   // UNICODE_TO_GBK[2130] := 16#4F5C;
   // UNICODE_TO_GBK[2131] := 16#D7F7;
   // UNICODE_TO_GBK[2132] := 16#4F5D;
   // UNICODE_TO_GBK[2133] := 16#D8FE;
   // UNICODE_TO_GBK[2134] := 16#4F5E;
   // UNICODE_TO_GBK[2135] := 16#D8FA;
   // UNICODE_TO_GBK[2136] := 16#4F5F;
   // UNICODE_TO_GBK[2137] := 16#D9A1;
   // UNICODE_TO_GBK[2138] := 16#4F60;
   // UNICODE_TO_GBK[2139] := 16#C4E3;
   // UNICODE_TO_GBK[2140] := 16#4F61;
   // UNICODE_TO_GBK[2141] := 16#81D9;
   // UNICODE_TO_GBK[2142] := 16#4F62;
   // UNICODE_TO_GBK[2143] := 16#81DA;
   // UNICODE_TO_GBK[2144] := 16#4F63;
   // UNICODE_TO_GBK[2145] := 16#D3B6;
   // UNICODE_TO_GBK[2146] := 16#4F64;
   // UNICODE_TO_GBK[2147] := 16#D8F4;
   // UNICODE_TO_GBK[2148] := 16#4F65;
   // UNICODE_TO_GBK[2149] := 16#D9DD;
   // UNICODE_TO_GBK[2150] := 16#4F66;
   // UNICODE_TO_GBK[2151] := 16#81DB;
   // UNICODE_TO_GBK[2152] := 16#4F67;
   // UNICODE_TO_GBK[2153] := 16#D8FB;
   // UNICODE_TO_GBK[2154] := 16#4F68;
   // UNICODE_TO_GBK[2155] := 16#81DC;
   // UNICODE_TO_GBK[2156] := 16#4F69;
   // UNICODE_TO_GBK[2157] := 16#C5E5;
   // UNICODE_TO_GBK[2158] := 16#4F6A;
   // UNICODE_TO_GBK[2159] := 16#81DD;
   // UNICODE_TO_GBK[2160] := 16#4F6B;
   // UNICODE_TO_GBK[2161] := 16#81DE;
   // UNICODE_TO_GBK[2162] := 16#4F6C;
   // UNICODE_TO_GBK[2163] := 16#C0D0;
   // UNICODE_TO_GBK[2164] := 16#4F6D;
   // UNICODE_TO_GBK[2165] := 16#81DF;
   // UNICODE_TO_GBK[2166] := 16#4F6E;
   // UNICODE_TO_GBK[2167] := 16#81E0;
   // UNICODE_TO_GBK[2168] := 16#4F6F;
   // UNICODE_TO_GBK[2169] := 16#D1F0;
   // UNICODE_TO_GBK[2170] := 16#4F70;
   // UNICODE_TO_GBK[2171] := 16#B0DB;
   // UNICODE_TO_GBK[2172] := 16#4F71;
   // UNICODE_TO_GBK[2173] := 16#81E1;
   // UNICODE_TO_GBK[2174] := 16#4F72;
   // UNICODE_TO_GBK[2175] := 16#81E2;
   // UNICODE_TO_GBK[2176] := 16#4F73;
   // UNICODE_TO_GBK[2177] := 16#BCD1;
   // UNICODE_TO_GBK[2178] := 16#4F74;
   // UNICODE_TO_GBK[2179] := 16#D9A6;
   // UNICODE_TO_GBK[2180] := 16#4F75;
   // UNICODE_TO_GBK[2181] := 16#81E3;
   // UNICODE_TO_GBK[2182] := 16#4F76;
   // UNICODE_TO_GBK[2183] := 16#D9A5;
   // UNICODE_TO_GBK[2184] := 16#4F77;
   // UNICODE_TO_GBK[2185] := 16#81E4;
   // UNICODE_TO_GBK[2186] := 16#4F78;
   // UNICODE_TO_GBK[2187] := 16#81E5;
   // UNICODE_TO_GBK[2188] := 16#4F79;
   // UNICODE_TO_GBK[2189] := 16#81E6;
   // UNICODE_TO_GBK[2190] := 16#4F7A;
   // UNICODE_TO_GBK[2191] := 16#81E7;
   // UNICODE_TO_GBK[2192] := 16#4F7B;
   // UNICODE_TO_GBK[2193] := 16#D9AC;
   // UNICODE_TO_GBK[2194] := 16#4F7C;
   // UNICODE_TO_GBK[2195] := 16#D9AE;
   // UNICODE_TO_GBK[2196] := 16#4F7D;
   // UNICODE_TO_GBK[2197] := 16#81E8;
   // UNICODE_TO_GBK[2198] := 16#4F7E;
   // UNICODE_TO_GBK[2199] := 16#D9AB;
   // UNICODE_TO_GBK[2200] := 16#4F7F;
   // UNICODE_TO_GBK[2201] := 16#CAB9;
   // UNICODE_TO_GBK[2202] := 16#4F80;
   // UNICODE_TO_GBK[2203] := 16#81E9;
   // UNICODE_TO_GBK[2204] := 16#4F81;
   // UNICODE_TO_GBK[2205] := 16#81EA;
   // UNICODE_TO_GBK[2206] := 16#4F82;
   // UNICODE_TO_GBK[2207] := 16#81EB;
   // UNICODE_TO_GBK[2208] := 16#4F83;
   // UNICODE_TO_GBK[2209] := 16#D9A9;
   // UNICODE_TO_GBK[2210] := 16#4F84;
   // UNICODE_TO_GBK[2211] := 16#D6B6;
   // UNICODE_TO_GBK[2212] := 16#4F85;
   // UNICODE_TO_GBK[2213] := 16#81EC;
   // UNICODE_TO_GBK[2214] := 16#4F86;
   // UNICODE_TO_GBK[2215] := 16#81ED;
   // UNICODE_TO_GBK[2216] := 16#4F87;
   // UNICODE_TO_GBK[2217] := 16#81EE;
   // UNICODE_TO_GBK[2218] := 16#4F88;
   // UNICODE_TO_GBK[2219] := 16#B3DE;
   // UNICODE_TO_GBK[2220] := 16#4F89;
   // UNICODE_TO_GBK[2221] := 16#D9A8;
   // UNICODE_TO_GBK[2222] := 16#4F8A;
   // UNICODE_TO_GBK[2223] := 16#81EF;
   // UNICODE_TO_GBK[2224] := 16#4F8B;
   // UNICODE_TO_GBK[2225] := 16#C0FD;
   // UNICODE_TO_GBK[2226] := 16#4F8C;
   // UNICODE_TO_GBK[2227] := 16#81F0;
   // UNICODE_TO_GBK[2228] := 16#4F8D;
   // UNICODE_TO_GBK[2229] := 16#CACC;
   // UNICODE_TO_GBK[2230] := 16#4F8E;
   // UNICODE_TO_GBK[2231] := 16#81F1;
   // UNICODE_TO_GBK[2232] := 16#4F8F;
   // UNICODE_TO_GBK[2233] := 16#D9AA;
   // UNICODE_TO_GBK[2234] := 16#4F90;
   // UNICODE_TO_GBK[2235] := 16#81F2;
   // UNICODE_TO_GBK[2236] := 16#4F91;
   // UNICODE_TO_GBK[2237] := 16#D9A7;
   // UNICODE_TO_GBK[2238] := 16#4F92;
   // UNICODE_TO_GBK[2239] := 16#81F3;
   // UNICODE_TO_GBK[2240] := 16#4F93;
   // UNICODE_TO_GBK[2241] := 16#81F4;
   // UNICODE_TO_GBK[2242] := 16#4F94;
   // UNICODE_TO_GBK[2243] := 16#D9B0;
   // UNICODE_TO_GBK[2244] := 16#4F95;
   // UNICODE_TO_GBK[2245] := 16#81F5;
   // UNICODE_TO_GBK[2246] := 16#4F96;
   // UNICODE_TO_GBK[2247] := 16#81F6;
   // UNICODE_TO_GBK[2248] := 16#4F97;
   // UNICODE_TO_GBK[2249] := 16#B6B1;
   // UNICODE_TO_GBK[2250] := 16#4F98;
   // UNICODE_TO_GBK[2251] := 16#81F7;
   // UNICODE_TO_GBK[2252] := 16#4F99;
   // UNICODE_TO_GBK[2253] := 16#81F8;
   // UNICODE_TO_GBK[2254] := 16#4F9A;
   // UNICODE_TO_GBK[2255] := 16#81F9;
   // UNICODE_TO_GBK[2256] := 16#4F9B;
   // UNICODE_TO_GBK[2257] := 16#B9A9;
   // UNICODE_TO_GBK[2258] := 16#4F9C;
   // UNICODE_TO_GBK[2259] := 16#81FA;
   // UNICODE_TO_GBK[2260] := 16#4F9D;
   // UNICODE_TO_GBK[2261] := 16#D2C0;
   // UNICODE_TO_GBK[2262] := 16#4F9E;
   // UNICODE_TO_GBK[2263] := 16#81FB;
   // UNICODE_TO_GBK[2264] := 16#4F9F;
   // UNICODE_TO_GBK[2265] := 16#81FC;
   // UNICODE_TO_GBK[2266] := 16#4FA0;
   // UNICODE_TO_GBK[2267] := 16#CFC0;
   // UNICODE_TO_GBK[2268] := 16#4FA1;
   // UNICODE_TO_GBK[2269] := 16#81FD;
   // UNICODE_TO_GBK[2270] := 16#4FA2;
   // UNICODE_TO_GBK[2271] := 16#81FE;
   // UNICODE_TO_GBK[2272] := 16#4FA3;
   // UNICODE_TO_GBK[2273] := 16#C2C2;
   // UNICODE_TO_GBK[2274] := 16#4FA4;
   // UNICODE_TO_GBK[2275] := 16#8240;
   // UNICODE_TO_GBK[2276] := 16#4FA5;
   // UNICODE_TO_GBK[2277] := 16#BDC4;
   // UNICODE_TO_GBK[2278] := 16#4FA6;
   // UNICODE_TO_GBK[2279] := 16#D5EC;
   // UNICODE_TO_GBK[2280] := 16#4FA7;
   // UNICODE_TO_GBK[2281] := 16#B2E0;
   // UNICODE_TO_GBK[2282] := 16#4FA8;
   // UNICODE_TO_GBK[2283] := 16#C7C8;
   // UNICODE_TO_GBK[2284] := 16#4FA9;
   // UNICODE_TO_GBK[2285] := 16#BFEB;
   // UNICODE_TO_GBK[2286] := 16#4FAA;
   // UNICODE_TO_GBK[2287] := 16#D9AD;
   // UNICODE_TO_GBK[2288] := 16#4FAB;
   // UNICODE_TO_GBK[2289] := 16#8241;
   // UNICODE_TO_GBK[2290] := 16#4FAC;
   // UNICODE_TO_GBK[2291] := 16#D9AF;
   // UNICODE_TO_GBK[2292] := 16#4FAD;
   // UNICODE_TO_GBK[2293] := 16#8242;
   // UNICODE_TO_GBK[2294] := 16#4FAE;
   // UNICODE_TO_GBK[2295] := 16#CEEA;
   // UNICODE_TO_GBK[2296] := 16#4FAF;
   // UNICODE_TO_GBK[2297] := 16#BAEE;
   // UNICODE_TO_GBK[2298] := 16#4FB0;
   // UNICODE_TO_GBK[2299] := 16#8243;
   // UNICODE_TO_GBK[2300] := 16#4FB1;
   // UNICODE_TO_GBK[2301] := 16#8244;
   // UNICODE_TO_GBK[2302] := 16#4FB2;
   // UNICODE_TO_GBK[2303] := 16#8245;
   // UNICODE_TO_GBK[2304] := 16#4FB3;
   // UNICODE_TO_GBK[2305] := 16#8246;
   // UNICODE_TO_GBK[2306] := 16#4FB4;
   // UNICODE_TO_GBK[2307] := 16#8247;
   // UNICODE_TO_GBK[2308] := 16#4FB5;
   // UNICODE_TO_GBK[2309] := 16#C7D6;
   // UNICODE_TO_GBK[2310] := 16#4FB6;
   // UNICODE_TO_GBK[2311] := 16#8248;
   // UNICODE_TO_GBK[2312] := 16#4FB7;
   // UNICODE_TO_GBK[2313] := 16#8249;
   // UNICODE_TO_GBK[2314] := 16#4FB8;
   // UNICODE_TO_GBK[2315] := 16#824A;
   // UNICODE_TO_GBK[2316] := 16#4FB9;
   // UNICODE_TO_GBK[2317] := 16#824B;
   // UNICODE_TO_GBK[2318] := 16#4FBA;
   // UNICODE_TO_GBK[2319] := 16#824C;
   // UNICODE_TO_GBK[2320] := 16#4FBB;
   // UNICODE_TO_GBK[2321] := 16#824D;
   // UNICODE_TO_GBK[2322] := 16#4FBC;
   // UNICODE_TO_GBK[2323] := 16#824E;
   // UNICODE_TO_GBK[2324] := 16#4FBD;
   // UNICODE_TO_GBK[2325] := 16#824F;
   // UNICODE_TO_GBK[2326] := 16#4FBE;
   // UNICODE_TO_GBK[2327] := 16#8250;
   // UNICODE_TO_GBK[2328] := 16#4FBF;
   // UNICODE_TO_GBK[2329] := 16#B1E3;
   // UNICODE_TO_GBK[2330] := 16#4FC0;
   // UNICODE_TO_GBK[2331] := 16#8251;
   // UNICODE_TO_GBK[2332] := 16#4FC1;
   // UNICODE_TO_GBK[2333] := 16#8252;
   // UNICODE_TO_GBK[2334] := 16#4FC2;
   // UNICODE_TO_GBK[2335] := 16#8253;
   // UNICODE_TO_GBK[2336] := 16#4FC3;
   // UNICODE_TO_GBK[2337] := 16#B4D9;
   // UNICODE_TO_GBK[2338] := 16#4FC4;
   // UNICODE_TO_GBK[2339] := 16#B6ED;
   // UNICODE_TO_GBK[2340] := 16#4FC5;
   // UNICODE_TO_GBK[2341] := 16#D9B4;
   // UNICODE_TO_GBK[2342] := 16#4FC6;
   // UNICODE_TO_GBK[2343] := 16#8254;
   // UNICODE_TO_GBK[2344] := 16#4FC7;
   // UNICODE_TO_GBK[2345] := 16#8255;
   // UNICODE_TO_GBK[2346] := 16#4FC8;
   // UNICODE_TO_GBK[2347] := 16#8256;
   // UNICODE_TO_GBK[2348] := 16#4FC9;
   // UNICODE_TO_GBK[2349] := 16#8257;
   // UNICODE_TO_GBK[2350] := 16#4FCA;
   // UNICODE_TO_GBK[2351] := 16#BFA1;
   // UNICODE_TO_GBK[2352] := 16#4FCB;
   // UNICODE_TO_GBK[2353] := 16#8258;
   // UNICODE_TO_GBK[2354] := 16#4FCC;
   // UNICODE_TO_GBK[2355] := 16#8259;
   // UNICODE_TO_GBK[2356] := 16#4FCD;
   // UNICODE_TO_GBK[2357] := 16#825A;
   // UNICODE_TO_GBK[2358] := 16#4FCE;
   // UNICODE_TO_GBK[2359] := 16#D9DE;
   // UNICODE_TO_GBK[2360] := 16#4FCF;
   // UNICODE_TO_GBK[2361] := 16#C7CE;
   // UNICODE_TO_GBK[2362] := 16#4FD0;
   // UNICODE_TO_GBK[2363] := 16#C0FE;
   // UNICODE_TO_GBK[2364] := 16#4FD1;
   // UNICODE_TO_GBK[2365] := 16#D9B8;
   // UNICODE_TO_GBK[2366] := 16#4FD2;
   // UNICODE_TO_GBK[2367] := 16#825B;
   // UNICODE_TO_GBK[2368] := 16#4FD3;
   // UNICODE_TO_GBK[2369] := 16#825C;
   // UNICODE_TO_GBK[2370] := 16#4FD4;
   // UNICODE_TO_GBK[2371] := 16#825D;
   // UNICODE_TO_GBK[2372] := 16#4FD5;
   // UNICODE_TO_GBK[2373] := 16#825E;
   // UNICODE_TO_GBK[2374] := 16#4FD6;
   // UNICODE_TO_GBK[2375] := 16#825F;
   // UNICODE_TO_GBK[2376] := 16#4FD7;
   // UNICODE_TO_GBK[2377] := 16#CBD7;
   // UNICODE_TO_GBK[2378] := 16#4FD8;
   // UNICODE_TO_GBK[2379] := 16#B7FD;
   // UNICODE_TO_GBK[2380] := 16#4FD9;
   // UNICODE_TO_GBK[2381] := 16#8260;
   // UNICODE_TO_GBK[2382] := 16#4FDA;
   // UNICODE_TO_GBK[2383] := 16#D9B5;
   // UNICODE_TO_GBK[2384] := 16#4FDB;
   // UNICODE_TO_GBK[2385] := 16#8261;
   // UNICODE_TO_GBK[2386] := 16#4FDC;
   // UNICODE_TO_GBK[2387] := 16#D9B7;
   // UNICODE_TO_GBK[2388] := 16#4FDD;
   // UNICODE_TO_GBK[2389] := 16#B1A3;
   // UNICODE_TO_GBK[2390] := 16#4FDE;
   // UNICODE_TO_GBK[2391] := 16#D3E1;
   // UNICODE_TO_GBK[2392] := 16#4FDF;
   // UNICODE_TO_GBK[2393] := 16#D9B9;
   // UNICODE_TO_GBK[2394] := 16#4FE0;
   // UNICODE_TO_GBK[2395] := 16#8262;
   // UNICODE_TO_GBK[2396] := 16#4FE1;
   // UNICODE_TO_GBK[2397] := 16#D0C5;
   // UNICODE_TO_GBK[2398] := 16#4FE2;
   // UNICODE_TO_GBK[2399] := 16#8263;
   // UNICODE_TO_GBK[2400] := 16#4FE3;
   // UNICODE_TO_GBK[2401] := 16#D9B6;
   // UNICODE_TO_GBK[2402] := 16#4FE4;
   // UNICODE_TO_GBK[2403] := 16#8264;
   // UNICODE_TO_GBK[2404] := 16#4FE5;
   // UNICODE_TO_GBK[2405] := 16#8265;
   // UNICODE_TO_GBK[2406] := 16#4FE6;
   // UNICODE_TO_GBK[2407] := 16#D9B1;
   // UNICODE_TO_GBK[2408] := 16#4FE7;
   // UNICODE_TO_GBK[2409] := 16#8266;
   // UNICODE_TO_GBK[2410] := 16#4FE8;
   // UNICODE_TO_GBK[2411] := 16#D9B2;
   // UNICODE_TO_GBK[2412] := 16#4FE9;
   // UNICODE_TO_GBK[2413] := 16#C1A9;
   // UNICODE_TO_GBK[2414] := 16#4FEA;
   // UNICODE_TO_GBK[2415] := 16#D9B3;
   // UNICODE_TO_GBK[2416] := 16#4FEB;
   // UNICODE_TO_GBK[2417] := 16#8267;
   // UNICODE_TO_GBK[2418] := 16#4FEC;
   // UNICODE_TO_GBK[2419] := 16#8268;
   // UNICODE_TO_GBK[2420] := 16#4FED;
   // UNICODE_TO_GBK[2421] := 16#BCF3;
   // UNICODE_TO_GBK[2422] := 16#4FEE;
   // UNICODE_TO_GBK[2423] := 16#D0DE;
   // UNICODE_TO_GBK[2424] := 16#4FEF;
   // UNICODE_TO_GBK[2425] := 16#B8A9;
   // UNICODE_TO_GBK[2426] := 16#4FF0;
   // UNICODE_TO_GBK[2427] := 16#8269;
   // UNICODE_TO_GBK[2428] := 16#4FF1;
   // UNICODE_TO_GBK[2429] := 16#BEE3;
   // UNICODE_TO_GBK[2430] := 16#4FF2;
   // UNICODE_TO_GBK[2431] := 16#826A;
   // UNICODE_TO_GBK[2432] := 16#4FF3;
   // UNICODE_TO_GBK[2433] := 16#D9BD;
   // UNICODE_TO_GBK[2434] := 16#4FF4;
   // UNICODE_TO_GBK[2435] := 16#826B;
   // UNICODE_TO_GBK[2436] := 16#4FF5;
   // UNICODE_TO_GBK[2437] := 16#826C;
   // UNICODE_TO_GBK[2438] := 16#4FF6;
   // UNICODE_TO_GBK[2439] := 16#826D;
   // UNICODE_TO_GBK[2440] := 16#4FF7;
   // UNICODE_TO_GBK[2441] := 16#826E;
   // UNICODE_TO_GBK[2442] := 16#4FF8;
   // UNICODE_TO_GBK[2443] := 16#D9BA;
   // UNICODE_TO_GBK[2444] := 16#4FF9;
   // UNICODE_TO_GBK[2445] := 16#826F;
   // UNICODE_TO_GBK[2446] := 16#4FFA;
   // UNICODE_TO_GBK[2447] := 16#B0B3;
   // UNICODE_TO_GBK[2448] := 16#4FFB;
   // UNICODE_TO_GBK[2449] := 16#8270;
   // UNICODE_TO_GBK[2450] := 16#4FFC;
   // UNICODE_TO_GBK[2451] := 16#8271;
   // UNICODE_TO_GBK[2452] := 16#4FFD;
   // UNICODE_TO_GBK[2453] := 16#8272;
   // UNICODE_TO_GBK[2454] := 16#4FFE;
   // UNICODE_TO_GBK[2455] := 16#D9C2;
   // UNICODE_TO_GBK[2456] := 16#4FFF;
   // UNICODE_TO_GBK[2457] := 16#8273;
   // UNICODE_TO_GBK[2458] := 16#5000;
   // UNICODE_TO_GBK[2459] := 16#8274;
   // UNICODE_TO_GBK[2460] := 16#5001;
   // UNICODE_TO_GBK[2461] := 16#8275;
   // UNICODE_TO_GBK[2462] := 16#5002;
   // UNICODE_TO_GBK[2463] := 16#8276;
   // UNICODE_TO_GBK[2464] := 16#5003;
   // UNICODE_TO_GBK[2465] := 16#8277;
   // UNICODE_TO_GBK[2466] := 16#5004;
   // UNICODE_TO_GBK[2467] := 16#8278;
   // UNICODE_TO_GBK[2468] := 16#5005;
   // UNICODE_TO_GBK[2469] := 16#8279;
   // UNICODE_TO_GBK[2470] := 16#5006;
   // UNICODE_TO_GBK[2471] := 16#827A;
   // UNICODE_TO_GBK[2472] := 16#5007;
   // UNICODE_TO_GBK[2473] := 16#827B;
   // UNICODE_TO_GBK[2474] := 16#5008;
   // UNICODE_TO_GBK[2475] := 16#827C;
   // UNICODE_TO_GBK[2476] := 16#5009;
   // UNICODE_TO_GBK[2477] := 16#827D;
   // UNICODE_TO_GBK[2478] := 16#500A;
   // UNICODE_TO_GBK[2479] := 16#827E;
   // UNICODE_TO_GBK[2480] := 16#500B;
   // UNICODE_TO_GBK[2481] := 16#8280;
   // UNICODE_TO_GBK[2482] := 16#500C;
   // UNICODE_TO_GBK[2483] := 16#D9C4;
   // UNICODE_TO_GBK[2484] := 16#500D;
   // UNICODE_TO_GBK[2485] := 16#B1B6;
   // UNICODE_TO_GBK[2486] := 16#500E;
   // UNICODE_TO_GBK[2487] := 16#8281;
   // UNICODE_TO_GBK[2488] := 16#500F;
   // UNICODE_TO_GBK[2489] := 16#D9BF;
   // UNICODE_TO_GBK[2490] := 16#5010;
   // UNICODE_TO_GBK[2491] := 16#8282;
   // UNICODE_TO_GBK[2492] := 16#5011;
   // UNICODE_TO_GBK[2493] := 16#8283;
   // UNICODE_TO_GBK[2494] := 16#5012;
   // UNICODE_TO_GBK[2495] := 16#B5B9;
   // UNICODE_TO_GBK[2496] := 16#5013;
   // UNICODE_TO_GBK[2497] := 16#8284;
   // UNICODE_TO_GBK[2498] := 16#5014;
   // UNICODE_TO_GBK[2499] := 16#BEF3;
   // UNICODE_TO_GBK[2500] := 16#5015;
   // UNICODE_TO_GBK[2501] := 16#8285;
   // UNICODE_TO_GBK[2502] := 16#5016;
   // UNICODE_TO_GBK[2503] := 16#8286;
   // UNICODE_TO_GBK[2504] := 16#5017;
   // UNICODE_TO_GBK[2505] := 16#8287;
   // UNICODE_TO_GBK[2506] := 16#5018;
   // UNICODE_TO_GBK[2507] := 16#CCC8;
   // UNICODE_TO_GBK[2508] := 16#5019;
   // UNICODE_TO_GBK[2509] := 16#BAF2;
   // UNICODE_TO_GBK[2510] := 16#501A;
   // UNICODE_TO_GBK[2511] := 16#D2D0;
   // UNICODE_TO_GBK[2512] := 16#501B;
   // UNICODE_TO_GBK[2513] := 16#8288;
   // UNICODE_TO_GBK[2514] := 16#501C;
   // UNICODE_TO_GBK[2515] := 16#D9C3;
   // UNICODE_TO_GBK[2516] := 16#501D;
   // UNICODE_TO_GBK[2517] := 16#8289;
   // UNICODE_TO_GBK[2518] := 16#501E;
   // UNICODE_TO_GBK[2519] := 16#828A;
   // UNICODE_TO_GBK[2520] := 16#501F;
   // UNICODE_TO_GBK[2521] := 16#BDE8;
   // UNICODE_TO_GBK[2522] := 16#5020;
   // UNICODE_TO_GBK[2523] := 16#828B;
   // UNICODE_TO_GBK[2524] := 16#5021;
   // UNICODE_TO_GBK[2525] := 16#B3AB;
   // UNICODE_TO_GBK[2526] := 16#5022;
   // UNICODE_TO_GBK[2527] := 16#828C;
   // UNICODE_TO_GBK[2528] := 16#5023;
   // UNICODE_TO_GBK[2529] := 16#828D;
   // UNICODE_TO_GBK[2530] := 16#5024;
   // UNICODE_TO_GBK[2531] := 16#828E;
   // UNICODE_TO_GBK[2532] := 16#5025;
   // UNICODE_TO_GBK[2533] := 16#D9C5;
   // UNICODE_TO_GBK[2534] := 16#5026;
   // UNICODE_TO_GBK[2535] := 16#BEEB;
   // UNICODE_TO_GBK[2536] := 16#5027;
   // UNICODE_TO_GBK[2537] := 16#828F;
   // UNICODE_TO_GBK[2538] := 16#5028;
   // UNICODE_TO_GBK[2539] := 16#D9C6;
   // UNICODE_TO_GBK[2540] := 16#5029;
   // UNICODE_TO_GBK[2541] := 16#D9BB;
   // UNICODE_TO_GBK[2542] := 16#502A;
   // UNICODE_TO_GBK[2543] := 16#C4DF;
   // UNICODE_TO_GBK[2544] := 16#502B;
   // UNICODE_TO_GBK[2545] := 16#8290;
   // UNICODE_TO_GBK[2546] := 16#502C;
   // UNICODE_TO_GBK[2547] := 16#D9BE;
   // UNICODE_TO_GBK[2548] := 16#502D;
   // UNICODE_TO_GBK[2549] := 16#D9C1;
   // UNICODE_TO_GBK[2550] := 16#502E;
   // UNICODE_TO_GBK[2551] := 16#D9C0;
   // UNICODE_TO_GBK[2552] := 16#502F;
   // UNICODE_TO_GBK[2553] := 16#8291;
   // UNICODE_TO_GBK[2554] := 16#5030;
   // UNICODE_TO_GBK[2555] := 16#8292;
   // UNICODE_TO_GBK[2556] := 16#5031;
   // UNICODE_TO_GBK[2557] := 16#8293;
   // UNICODE_TO_GBK[2558] := 16#5032;
   // UNICODE_TO_GBK[2559] := 16#8294;
   // UNICODE_TO_GBK[2560] := 16#5033;
   // UNICODE_TO_GBK[2561] := 16#8295;
   // UNICODE_TO_GBK[2562] := 16#5034;
   // UNICODE_TO_GBK[2563] := 16#8296;
   // UNICODE_TO_GBK[2564] := 16#5035;
   // UNICODE_TO_GBK[2565] := 16#8297;
   // UNICODE_TO_GBK[2566] := 16#5036;
   // UNICODE_TO_GBK[2567] := 16#8298;
   // UNICODE_TO_GBK[2568] := 16#5037;
   // UNICODE_TO_GBK[2569] := 16#8299;
   // UNICODE_TO_GBK[2570] := 16#5038;
   // UNICODE_TO_GBK[2571] := 16#829A;
   // UNICODE_TO_GBK[2572] := 16#5039;
   // UNICODE_TO_GBK[2573] := 16#829B;
   // UNICODE_TO_GBK[2574] := 16#503A;
   // UNICODE_TO_GBK[2575] := 16#D5AE;
   // UNICODE_TO_GBK[2576] := 16#503B;
   // UNICODE_TO_GBK[2577] := 16#829C;
   // UNICODE_TO_GBK[2578] := 16#503C;
   // UNICODE_TO_GBK[2579] := 16#D6B5;
   // UNICODE_TO_GBK[2580] := 16#503D;
   // UNICODE_TO_GBK[2581] := 16#829D;
   // UNICODE_TO_GBK[2582] := 16#503E;
   // UNICODE_TO_GBK[2583] := 16#C7E3;
   // UNICODE_TO_GBK[2584] := 16#503F;
   // UNICODE_TO_GBK[2585] := 16#829E;
   // UNICODE_TO_GBK[2586] := 16#5040;
   // UNICODE_TO_GBK[2587] := 16#829F;
   // UNICODE_TO_GBK[2588] := 16#5041;
   // UNICODE_TO_GBK[2589] := 16#82A0;
   // UNICODE_TO_GBK[2590] := 16#5042;
   // UNICODE_TO_GBK[2591] := 16#82A1;
   // UNICODE_TO_GBK[2592] := 16#5043;
   // UNICODE_TO_GBK[2593] := 16#D9C8;
   // UNICODE_TO_GBK[2594] := 16#5044;
   // UNICODE_TO_GBK[2595] := 16#82A2;
   // UNICODE_TO_GBK[2596] := 16#5045;
   // UNICODE_TO_GBK[2597] := 16#82A3;
   // UNICODE_TO_GBK[2598] := 16#5046;
   // UNICODE_TO_GBK[2599] := 16#82A4;
   // UNICODE_TO_GBK[2600] := 16#5047;
   // UNICODE_TO_GBK[2601] := 16#BCD9;
   // UNICODE_TO_GBK[2602] := 16#5048;
   // UNICODE_TO_GBK[2603] := 16#D9CA;
   // UNICODE_TO_GBK[2604] := 16#5049;
   // UNICODE_TO_GBK[2605] := 16#82A5;
   // UNICODE_TO_GBK[2606] := 16#504A;
   // UNICODE_TO_GBK[2607] := 16#82A6;
   // UNICODE_TO_GBK[2608] := 16#504B;
   // UNICODE_TO_GBK[2609] := 16#82A7;
   // UNICODE_TO_GBK[2610] := 16#504C;
   // UNICODE_TO_GBK[2611] := 16#D9BC;
   // UNICODE_TO_GBK[2612] := 16#504D;
   // UNICODE_TO_GBK[2613] := 16#82A8;
   // UNICODE_TO_GBK[2614] := 16#504E;
   // UNICODE_TO_GBK[2615] := 16#D9CB;
   // UNICODE_TO_GBK[2616] := 16#504F;
   // UNICODE_TO_GBK[2617] := 16#C6AB;
   // UNICODE_TO_GBK[2618] := 16#5050;
   // UNICODE_TO_GBK[2619] := 16#82A9;
   // UNICODE_TO_GBK[2620] := 16#5051;
   // UNICODE_TO_GBK[2621] := 16#82AA;
   // UNICODE_TO_GBK[2622] := 16#5052;
   // UNICODE_TO_GBK[2623] := 16#82AB;
   // UNICODE_TO_GBK[2624] := 16#5053;
   // UNICODE_TO_GBK[2625] := 16#82AC;
   // UNICODE_TO_GBK[2626] := 16#5054;
   // UNICODE_TO_GBK[2627] := 16#82AD;
   // UNICODE_TO_GBK[2628] := 16#5055;
   // UNICODE_TO_GBK[2629] := 16#D9C9;
   // UNICODE_TO_GBK[2630] := 16#5056;
   // UNICODE_TO_GBK[2631] := 16#82AE;
   // UNICODE_TO_GBK[2632] := 16#5057;
   // UNICODE_TO_GBK[2633] := 16#82AF;
   // UNICODE_TO_GBK[2634] := 16#5058;
   // UNICODE_TO_GBK[2635] := 16#82B0;
   // UNICODE_TO_GBK[2636] := 16#5059;
   // UNICODE_TO_GBK[2637] := 16#82B1;
   // UNICODE_TO_GBK[2638] := 16#505A;
   // UNICODE_TO_GBK[2639] := 16#D7F6;
   // UNICODE_TO_GBK[2640] := 16#505B;
   // UNICODE_TO_GBK[2641] := 16#82B2;
   // UNICODE_TO_GBK[2642] := 16#505C;
   // UNICODE_TO_GBK[2643] := 16#CDA3;
   // UNICODE_TO_GBK[2644] := 16#505D;
   // UNICODE_TO_GBK[2645] := 16#82B3;
   // UNICODE_TO_GBK[2646] := 16#505E;
   // UNICODE_TO_GBK[2647] := 16#82B4;
   // UNICODE_TO_GBK[2648] := 16#505F;
   // UNICODE_TO_GBK[2649] := 16#82B5;
   // UNICODE_TO_GBK[2650] := 16#5060;
   // UNICODE_TO_GBK[2651] := 16#82B6;
   // UNICODE_TO_GBK[2652] := 16#5061;
   // UNICODE_TO_GBK[2653] := 16#82B7;
   // UNICODE_TO_GBK[2654] := 16#5062;
   // UNICODE_TO_GBK[2655] := 16#82B8;
   // UNICODE_TO_GBK[2656] := 16#5063;
   // UNICODE_TO_GBK[2657] := 16#82B9;
   // UNICODE_TO_GBK[2658] := 16#5064;
   // UNICODE_TO_GBK[2659] := 16#82BA;
   // UNICODE_TO_GBK[2660] := 16#5065;
   // UNICODE_TO_GBK[2661] := 16#BDA1;
   // UNICODE_TO_GBK[2662] := 16#5066;
   // UNICODE_TO_GBK[2663] := 16#82BB;
   // UNICODE_TO_GBK[2664] := 16#5067;
   // UNICODE_TO_GBK[2665] := 16#82BC;
   // UNICODE_TO_GBK[2666] := 16#5068;
   // UNICODE_TO_GBK[2667] := 16#82BD;
   // UNICODE_TO_GBK[2668] := 16#5069;
   // UNICODE_TO_GBK[2669] := 16#82BE;
   // UNICODE_TO_GBK[2670] := 16#506A;
   // UNICODE_TO_GBK[2671] := 16#82BF;
   // UNICODE_TO_GBK[2672] := 16#506B;
   // UNICODE_TO_GBK[2673] := 16#82C0;
   // UNICODE_TO_GBK[2674] := 16#506C;
   // UNICODE_TO_GBK[2675] := 16#D9CC;
   // UNICODE_TO_GBK[2676] := 16#506D;
   // UNICODE_TO_GBK[2677] := 16#82C1;
   // UNICODE_TO_GBK[2678] := 16#506E;
   // UNICODE_TO_GBK[2679] := 16#82C2;
   // UNICODE_TO_GBK[2680] := 16#506F;
   // UNICODE_TO_GBK[2681] := 16#82C3;
   // UNICODE_TO_GBK[2682] := 16#5070;
   // UNICODE_TO_GBK[2683] := 16#82C4;
   // UNICODE_TO_GBK[2684] := 16#5071;
   // UNICODE_TO_GBK[2685] := 16#82C5;
   // UNICODE_TO_GBK[2686] := 16#5072;
   // UNICODE_TO_GBK[2687] := 16#82C6;
   // UNICODE_TO_GBK[2688] := 16#5073;
   // UNICODE_TO_GBK[2689] := 16#82C7;
   // UNICODE_TO_GBK[2690] := 16#5074;
   // UNICODE_TO_GBK[2691] := 16#82C8;
   // UNICODE_TO_GBK[2692] := 16#5075;
   // UNICODE_TO_GBK[2693] := 16#82C9;
   // UNICODE_TO_GBK[2694] := 16#5076;
   // UNICODE_TO_GBK[2695] := 16#C5BC;
   // UNICODE_TO_GBK[2696] := 16#5077;
   // UNICODE_TO_GBK[2697] := 16#CDB5;
   // UNICODE_TO_GBK[2698] := 16#5078;
   // UNICODE_TO_GBK[2699] := 16#82CA;
   // UNICODE_TO_GBK[2700] := 16#5079;
   // UNICODE_TO_GBK[2701] := 16#82CB;
   // UNICODE_TO_GBK[2702] := 16#507A;
   // UNICODE_TO_GBK[2703] := 16#82CC;
   // UNICODE_TO_GBK[2704] := 16#507B;
   // UNICODE_TO_GBK[2705] := 16#D9CD;
   // UNICODE_TO_GBK[2706] := 16#507C;
   // UNICODE_TO_GBK[2707] := 16#82CD;
   // UNICODE_TO_GBK[2708] := 16#507D;
   // UNICODE_TO_GBK[2709] := 16#82CE;
   // UNICODE_TO_GBK[2710] := 16#507E;
   // UNICODE_TO_GBK[2711] := 16#D9C7;
   // UNICODE_TO_GBK[2712] := 16#507F;
   // UNICODE_TO_GBK[2713] := 16#B3A5;
   // UNICODE_TO_GBK[2714] := 16#5080;
   // UNICODE_TO_GBK[2715] := 16#BFFE;
   // UNICODE_TO_GBK[2716] := 16#5081;
   // UNICODE_TO_GBK[2717] := 16#82CF;
   // UNICODE_TO_GBK[2718] := 16#5082;
   // UNICODE_TO_GBK[2719] := 16#82D0;
   // UNICODE_TO_GBK[2720] := 16#5083;
   // UNICODE_TO_GBK[2721] := 16#82D1;
   // UNICODE_TO_GBK[2722] := 16#5084;
   // UNICODE_TO_GBK[2723] := 16#82D2;
   // UNICODE_TO_GBK[2724] := 16#5085;
   // UNICODE_TO_GBK[2725] := 16#B8B5;
   // UNICODE_TO_GBK[2726] := 16#5086;
   // UNICODE_TO_GBK[2727] := 16#82D3;
   // UNICODE_TO_GBK[2728] := 16#5087;
   // UNICODE_TO_GBK[2729] := 16#82D4;
   // UNICODE_TO_GBK[2730] := 16#5088;
   // UNICODE_TO_GBK[2731] := 16#C0FC;
   // UNICODE_TO_GBK[2732] := 16#5089;
   // UNICODE_TO_GBK[2733] := 16#82D5;
   // UNICODE_TO_GBK[2734] := 16#508A;
   // UNICODE_TO_GBK[2735] := 16#82D6;
   // UNICODE_TO_GBK[2736] := 16#508B;
   // UNICODE_TO_GBK[2737] := 16#82D7;
   // UNICODE_TO_GBK[2738] := 16#508C;
   // UNICODE_TO_GBK[2739] := 16#82D8;
   // UNICODE_TO_GBK[2740] := 16#508D;
   // UNICODE_TO_GBK[2741] := 16#B0F8;
   // UNICODE_TO_GBK[2742] := 16#508E;
   // UNICODE_TO_GBK[2743] := 16#82D9;
   // UNICODE_TO_GBK[2744] := 16#508F;
   // UNICODE_TO_GBK[2745] := 16#82DA;
   // UNICODE_TO_GBK[2746] := 16#5090;
   // UNICODE_TO_GBK[2747] := 16#82DB;
   // UNICODE_TO_GBK[2748] := 16#5091;
   // UNICODE_TO_GBK[2749] := 16#82DC;
   // UNICODE_TO_GBK[2750] := 16#5092;
   // UNICODE_TO_GBK[2751] := 16#82DD;
   // UNICODE_TO_GBK[2752] := 16#5093;
   // UNICODE_TO_GBK[2753] := 16#82DE;
   // UNICODE_TO_GBK[2754] := 16#5094;
   // UNICODE_TO_GBK[2755] := 16#82DF;
   // UNICODE_TO_GBK[2756] := 16#5095;
   // UNICODE_TO_GBK[2757] := 16#82E0;
   // UNICODE_TO_GBK[2758] := 16#5096;
   // UNICODE_TO_GBK[2759] := 16#82E1;
   // UNICODE_TO_GBK[2760] := 16#5097;
   // UNICODE_TO_GBK[2761] := 16#82E2;
   // UNICODE_TO_GBK[2762] := 16#5098;
   // UNICODE_TO_GBK[2763] := 16#82E3;
   // UNICODE_TO_GBK[2764] := 16#5099;
   // UNICODE_TO_GBK[2765] := 16#82E4;
   // UNICODE_TO_GBK[2766] := 16#509A;
   // UNICODE_TO_GBK[2767] := 16#82E5;
   // UNICODE_TO_GBK[2768] := 16#509B;
   // UNICODE_TO_GBK[2769] := 16#82E6;
   // UNICODE_TO_GBK[2770] := 16#509C;
   // UNICODE_TO_GBK[2771] := 16#82E7;
   // UNICODE_TO_GBK[2772] := 16#509D;
   // UNICODE_TO_GBK[2773] := 16#82E8;
   // UNICODE_TO_GBK[2774] := 16#509E;
   // UNICODE_TO_GBK[2775] := 16#82E9;
   // UNICODE_TO_GBK[2776] := 16#509F;
   // UNICODE_TO_GBK[2777] := 16#82EA;
   // UNICODE_TO_GBK[2778] := 16#50A0;
   // UNICODE_TO_GBK[2779] := 16#82EB;
   // UNICODE_TO_GBK[2780] := 16#50A1;
   // UNICODE_TO_GBK[2781] := 16#82EC;
   // UNICODE_TO_GBK[2782] := 16#50A2;
   // UNICODE_TO_GBK[2783] := 16#82ED;
   // UNICODE_TO_GBK[2784] := 16#50A3;
   // UNICODE_TO_GBK[2785] := 16#B4F6;
   // UNICODE_TO_GBK[2786] := 16#50A4;
   // UNICODE_TO_GBK[2787] := 16#82EE;
   // UNICODE_TO_GBK[2788] := 16#50A5;
   // UNICODE_TO_GBK[2789] := 16#D9CE;
   // UNICODE_TO_GBK[2790] := 16#50A6;
   // UNICODE_TO_GBK[2791] := 16#82EF;
   // UNICODE_TO_GBK[2792] := 16#50A7;
   // UNICODE_TO_GBK[2793] := 16#D9CF;
   // UNICODE_TO_GBK[2794] := 16#50A8;
   // UNICODE_TO_GBK[2795] := 16#B4A2;
   // UNICODE_TO_GBK[2796] := 16#50A9;
   // UNICODE_TO_GBK[2797] := 16#D9D0;
   // UNICODE_TO_GBK[2798] := 16#50AA;
   // UNICODE_TO_GBK[2799] := 16#82F0;
   // UNICODE_TO_GBK[2800] := 16#50AB;
   // UNICODE_TO_GBK[2801] := 16#82F1;
   // UNICODE_TO_GBK[2802] := 16#50AC;
   // UNICODE_TO_GBK[2803] := 16#B4DF;
   // UNICODE_TO_GBK[2804] := 16#50AD;
   // UNICODE_TO_GBK[2805] := 16#82F2;
   // UNICODE_TO_GBK[2806] := 16#50AE;
   // UNICODE_TO_GBK[2807] := 16#82F3;
   // UNICODE_TO_GBK[2808] := 16#50AF;
   // UNICODE_TO_GBK[2809] := 16#82F4;
   // UNICODE_TO_GBK[2810] := 16#50B0;
   // UNICODE_TO_GBK[2811] := 16#82F5;
   // UNICODE_TO_GBK[2812] := 16#50B1;
   // UNICODE_TO_GBK[2813] := 16#82F6;
   // UNICODE_TO_GBK[2814] := 16#50B2;
   // UNICODE_TO_GBK[2815] := 16#B0C1;
   // UNICODE_TO_GBK[2816] := 16#50B3;
   // UNICODE_TO_GBK[2817] := 16#82F7;
   // UNICODE_TO_GBK[2818] := 16#50B4;
   // UNICODE_TO_GBK[2819] := 16#82F8;
   // UNICODE_TO_GBK[2820] := 16#50B5;
   // UNICODE_TO_GBK[2821] := 16#82F9;
   // UNICODE_TO_GBK[2822] := 16#50B6;
   // UNICODE_TO_GBK[2823] := 16#82FA;
   // UNICODE_TO_GBK[2824] := 16#50B7;
   // UNICODE_TO_GBK[2825] := 16#82FB;
   // UNICODE_TO_GBK[2826] := 16#50B8;
   // UNICODE_TO_GBK[2827] := 16#82FC;
   // UNICODE_TO_GBK[2828] := 16#50B9;
   // UNICODE_TO_GBK[2829] := 16#82FD;
   // UNICODE_TO_GBK[2830] := 16#50BA;
   // UNICODE_TO_GBK[2831] := 16#D9D1;
   // UNICODE_TO_GBK[2832] := 16#50BB;
   // UNICODE_TO_GBK[2833] := 16#C9B5;
   // UNICODE_TO_GBK[2834] := 16#50BC;
   // UNICODE_TO_GBK[2835] := 16#82FE;
   // UNICODE_TO_GBK[2836] := 16#50BD;
   // UNICODE_TO_GBK[2837] := 16#8340;
   // UNICODE_TO_GBK[2838] := 16#50BE;
   // UNICODE_TO_GBK[2839] := 16#8341;
   // UNICODE_TO_GBK[2840] := 16#50BF;
   // UNICODE_TO_GBK[2841] := 16#8342;
   // UNICODE_TO_GBK[2842] := 16#50C0;
   // UNICODE_TO_GBK[2843] := 16#8343;
   // UNICODE_TO_GBK[2844] := 16#50C1;
   // UNICODE_TO_GBK[2845] := 16#8344;
   // UNICODE_TO_GBK[2846] := 16#50C2;
   // UNICODE_TO_GBK[2847] := 16#8345;
   // UNICODE_TO_GBK[2848] := 16#50C3;
   // UNICODE_TO_GBK[2849] := 16#8346;
   // UNICODE_TO_GBK[2850] := 16#50C4;
   // UNICODE_TO_GBK[2851] := 16#8347;
   // UNICODE_TO_GBK[2852] := 16#50C5;
   // UNICODE_TO_GBK[2853] := 16#8348;
   // UNICODE_TO_GBK[2854] := 16#50C6;
   // UNICODE_TO_GBK[2855] := 16#8349;
   // UNICODE_TO_GBK[2856] := 16#50C7;
   // UNICODE_TO_GBK[2857] := 16#834A;
   // UNICODE_TO_GBK[2858] := 16#50C8;
   // UNICODE_TO_GBK[2859] := 16#834B;
   // UNICODE_TO_GBK[2860] := 16#50C9;
   // UNICODE_TO_GBK[2861] := 16#834C;
   // UNICODE_TO_GBK[2862] := 16#50CA;
   // UNICODE_TO_GBK[2863] := 16#834D;
   // UNICODE_TO_GBK[2864] := 16#50CB;
   // UNICODE_TO_GBK[2865] := 16#834E;
   // UNICODE_TO_GBK[2866] := 16#50CC;
   // UNICODE_TO_GBK[2867] := 16#834F;
   // UNICODE_TO_GBK[2868] := 16#50CD;
   // UNICODE_TO_GBK[2869] := 16#8350;
   // UNICODE_TO_GBK[2870] := 16#50CE;
   // UNICODE_TO_GBK[2871] := 16#8351;
   // UNICODE_TO_GBK[2872] := 16#50CF;
   // UNICODE_TO_GBK[2873] := 16#CFF1;
   // UNICODE_TO_GBK[2874] := 16#50D0;
   // UNICODE_TO_GBK[2875] := 16#8352;
   // UNICODE_TO_GBK[2876] := 16#50D1;
   // UNICODE_TO_GBK[2877] := 16#8353;
   // UNICODE_TO_GBK[2878] := 16#50D2;
   // UNICODE_TO_GBK[2879] := 16#8354;
   // UNICODE_TO_GBK[2880] := 16#50D3;
   // UNICODE_TO_GBK[2881] := 16#8355;
   // UNICODE_TO_GBK[2882] := 16#50D4;
   // UNICODE_TO_GBK[2883] := 16#8356;
   // UNICODE_TO_GBK[2884] := 16#50D5;
   // UNICODE_TO_GBK[2885] := 16#8357;
   // UNICODE_TO_GBK[2886] := 16#50D6;
   // UNICODE_TO_GBK[2887] := 16#D9D2;
   // UNICODE_TO_GBK[2888] := 16#50D7;
   // UNICODE_TO_GBK[2889] := 16#8358;
   // UNICODE_TO_GBK[2890] := 16#50D8;
   // UNICODE_TO_GBK[2891] := 16#8359;
   // UNICODE_TO_GBK[2892] := 16#50D9;
   // UNICODE_TO_GBK[2893] := 16#835A;
   // UNICODE_TO_GBK[2894] := 16#50DA;
   // UNICODE_TO_GBK[2895] := 16#C1C5;
   // UNICODE_TO_GBK[2896] := 16#50DB;
   // UNICODE_TO_GBK[2897] := 16#835B;
   // UNICODE_TO_GBK[2898] := 16#50DC;
   // UNICODE_TO_GBK[2899] := 16#835C;
   // UNICODE_TO_GBK[2900] := 16#50DD;
   // UNICODE_TO_GBK[2901] := 16#835D;
   // UNICODE_TO_GBK[2902] := 16#50DE;
   // UNICODE_TO_GBK[2903] := 16#835E;
   // UNICODE_TO_GBK[2904] := 16#50DF;
   // UNICODE_TO_GBK[2905] := 16#835F;
   // UNICODE_TO_GBK[2906] := 16#50E0;
   // UNICODE_TO_GBK[2907] := 16#8360;
   // UNICODE_TO_GBK[2908] := 16#50E1;
   // UNICODE_TO_GBK[2909] := 16#8361;
   // UNICODE_TO_GBK[2910] := 16#50E2;
   // UNICODE_TO_GBK[2911] := 16#8362;
   // UNICODE_TO_GBK[2912] := 16#50E3;
   // UNICODE_TO_GBK[2913] := 16#8363;
   // UNICODE_TO_GBK[2914] := 16#50E4;
   // UNICODE_TO_GBK[2915] := 16#8364;
   // UNICODE_TO_GBK[2916] := 16#50E5;
   // UNICODE_TO_GBK[2917] := 16#8365;
   // UNICODE_TO_GBK[2918] := 16#50E6;
   // UNICODE_TO_GBK[2919] := 16#D9D6;
   // UNICODE_TO_GBK[2920] := 16#50E7;
   // UNICODE_TO_GBK[2921] := 16#C9AE;
   // UNICODE_TO_GBK[2922] := 16#50E8;
   // UNICODE_TO_GBK[2923] := 16#8366;
   // UNICODE_TO_GBK[2924] := 16#50E9;
   // UNICODE_TO_GBK[2925] := 16#8367;
   // UNICODE_TO_GBK[2926] := 16#50EA;
   // UNICODE_TO_GBK[2927] := 16#8368;
   // UNICODE_TO_GBK[2928] := 16#50EB;
   // UNICODE_TO_GBK[2929] := 16#8369;
   // UNICODE_TO_GBK[2930] := 16#50EC;
   // UNICODE_TO_GBK[2931] := 16#D9D5;
   // UNICODE_TO_GBK[2932] := 16#50ED;
   // UNICODE_TO_GBK[2933] := 16#D9D4;
   // UNICODE_TO_GBK[2934] := 16#50EE;
   // UNICODE_TO_GBK[2935] := 16#D9D7;
   // UNICODE_TO_GBK[2936] := 16#50EF;
   // UNICODE_TO_GBK[2937] := 16#836A;
   // UNICODE_TO_GBK[2938] := 16#50F0;
   // UNICODE_TO_GBK[2939] := 16#836B;
   // UNICODE_TO_GBK[2940] := 16#50F1;
   // UNICODE_TO_GBK[2941] := 16#836C;
   // UNICODE_TO_GBK[2942] := 16#50F2;
   // UNICODE_TO_GBK[2943] := 16#836D;
   // UNICODE_TO_GBK[2944] := 16#50F3;
   // UNICODE_TO_GBK[2945] := 16#CBDB;
   // UNICODE_TO_GBK[2946] := 16#50F4;
   // UNICODE_TO_GBK[2947] := 16#836E;
   // UNICODE_TO_GBK[2948] := 16#50F5;
   // UNICODE_TO_GBK[2949] := 16#BDA9;
   // UNICODE_TO_GBK[2950] := 16#50F6;
   // UNICODE_TO_GBK[2951] := 16#836F;
   // UNICODE_TO_GBK[2952] := 16#50F7;
   // UNICODE_TO_GBK[2953] := 16#8370;
   // UNICODE_TO_GBK[2954] := 16#50F8;
   // UNICODE_TO_GBK[2955] := 16#8371;
   // UNICODE_TO_GBK[2956] := 16#50F9;
   // UNICODE_TO_GBK[2957] := 16#8372;
   // UNICODE_TO_GBK[2958] := 16#50FA;
   // UNICODE_TO_GBK[2959] := 16#8373;
   // UNICODE_TO_GBK[2960] := 16#50FB;
   // UNICODE_TO_GBK[2961] := 16#C6A7;
   // UNICODE_TO_GBK[2962] := 16#50FC;
   // UNICODE_TO_GBK[2963] := 16#8374;
   // UNICODE_TO_GBK[2964] := 16#50FD;
   // UNICODE_TO_GBK[2965] := 16#8375;
   // UNICODE_TO_GBK[2966] := 16#50FE;
   // UNICODE_TO_GBK[2967] := 16#8376;
   // UNICODE_TO_GBK[2968] := 16#50FF;
   // UNICODE_TO_GBK[2969] := 16#8377;
   // UNICODE_TO_GBK[2970] := 16#5100;
   // UNICODE_TO_GBK[2971] := 16#8378;
   // UNICODE_TO_GBK[2972] := 16#5101;
   // UNICODE_TO_GBK[2973] := 16#8379;
   // UNICODE_TO_GBK[2974] := 16#5102;
   // UNICODE_TO_GBK[2975] := 16#837A;
   // UNICODE_TO_GBK[2976] := 16#5103;
   // UNICODE_TO_GBK[2977] := 16#837B;
   // UNICODE_TO_GBK[2978] := 16#5104;
   // UNICODE_TO_GBK[2979] := 16#837C;
   // UNICODE_TO_GBK[2980] := 16#5105;
   // UNICODE_TO_GBK[2981] := 16#837D;
   // UNICODE_TO_GBK[2982] := 16#5106;
   // UNICODE_TO_GBK[2983] := 16#D9D3;
   // UNICODE_TO_GBK[2984] := 16#5107;
   // UNICODE_TO_GBK[2985] := 16#D9D8;
   // UNICODE_TO_GBK[2986] := 16#5108;
   // UNICODE_TO_GBK[2987] := 16#837E;
   // UNICODE_TO_GBK[2988] := 16#5109;
   // UNICODE_TO_GBK[2989] := 16#8380;
   // UNICODE_TO_GBK[2990] := 16#510A;
   // UNICODE_TO_GBK[2991] := 16#8381;
   // UNICODE_TO_GBK[2992] := 16#510B;
   // UNICODE_TO_GBK[2993] := 16#D9D9;
   // UNICODE_TO_GBK[2994] := 16#510C;
   // UNICODE_TO_GBK[2995] := 16#8382;
   // UNICODE_TO_GBK[2996] := 16#510D;
   // UNICODE_TO_GBK[2997] := 16#8383;
   // UNICODE_TO_GBK[2998] := 16#510E;
   // UNICODE_TO_GBK[2999] := 16#8384;
   // UNICODE_TO_GBK[3000] := 16#510F;
   // UNICODE_TO_GBK[3001] := 16#8385;
   // UNICODE_TO_GBK[3002] := 16#5110;
   // UNICODE_TO_GBK[3003] := 16#8386;
   // UNICODE_TO_GBK[3004] := 16#5111;
   // UNICODE_TO_GBK[3005] := 16#8387;
   // UNICODE_TO_GBK[3006] := 16#5112;
   // UNICODE_TO_GBK[3007] := 16#C8E5;
   // UNICODE_TO_GBK[3008] := 16#5113;
   // UNICODE_TO_GBK[3009] := 16#8388;
   // UNICODE_TO_GBK[3010] := 16#5114;
   // UNICODE_TO_GBK[3011] := 16#8389;
   // UNICODE_TO_GBK[3012] := 16#5115;
   // UNICODE_TO_GBK[3013] := 16#838A;
   // UNICODE_TO_GBK[3014] := 16#5116;
   // UNICODE_TO_GBK[3015] := 16#838B;
   // UNICODE_TO_GBK[3016] := 16#5117;
   // UNICODE_TO_GBK[3017] := 16#838C;
   // UNICODE_TO_GBK[3018] := 16#5118;
   // UNICODE_TO_GBK[3019] := 16#838D;
   // UNICODE_TO_GBK[3020] := 16#5119;
   // UNICODE_TO_GBK[3021] := 16#838E;
   // UNICODE_TO_GBK[3022] := 16#511A;
   // UNICODE_TO_GBK[3023] := 16#838F;
   // UNICODE_TO_GBK[3024] := 16#511B;
   // UNICODE_TO_GBK[3025] := 16#8390;
   // UNICODE_TO_GBK[3026] := 16#511C;
   // UNICODE_TO_GBK[3027] := 16#8391;
   // UNICODE_TO_GBK[3028] := 16#511D;
   // UNICODE_TO_GBK[3029] := 16#8392;
   // UNICODE_TO_GBK[3030] := 16#511E;
   // UNICODE_TO_GBK[3031] := 16#8393;
   // UNICODE_TO_GBK[3032] := 16#511F;
   // UNICODE_TO_GBK[3033] := 16#8394;
   // UNICODE_TO_GBK[3034] := 16#5120;
   // UNICODE_TO_GBK[3035] := 16#8395;
   // UNICODE_TO_GBK[3036] := 16#5121;
   // UNICODE_TO_GBK[3037] := 16#C0DC;
   // UNICODE_TO_GBK[3038] := 16#5122;
   // UNICODE_TO_GBK[3039] := 16#8396;
   // UNICODE_TO_GBK[3040] := 16#5123;
   // UNICODE_TO_GBK[3041] := 16#8397;
   // UNICODE_TO_GBK[3042] := 16#5124;
   // UNICODE_TO_GBK[3043] := 16#8398;
   // UNICODE_TO_GBK[3044] := 16#5125;
   // UNICODE_TO_GBK[3045] := 16#8399;
   // UNICODE_TO_GBK[3046] := 16#5126;
   // UNICODE_TO_GBK[3047] := 16#839A;
   // UNICODE_TO_GBK[3048] := 16#5127;
   // UNICODE_TO_GBK[3049] := 16#839B;
   // UNICODE_TO_GBK[3050] := 16#5128;
   // UNICODE_TO_GBK[3051] := 16#839C;
   // UNICODE_TO_GBK[3052] := 16#5129;
   // UNICODE_TO_GBK[3053] := 16#839D;
   // UNICODE_TO_GBK[3054] := 16#512A;
   // UNICODE_TO_GBK[3055] := 16#839E;
   // UNICODE_TO_GBK[3056] := 16#512B;
   // UNICODE_TO_GBK[3057] := 16#839F;
   // UNICODE_TO_GBK[3058] := 16#512C;
   // UNICODE_TO_GBK[3059] := 16#83A0;
   // UNICODE_TO_GBK[3060] := 16#512D;
   // UNICODE_TO_GBK[3061] := 16#83A1;
   // UNICODE_TO_GBK[3062] := 16#512E;
   // UNICODE_TO_GBK[3063] := 16#83A2;
   // UNICODE_TO_GBK[3064] := 16#512F;
   // UNICODE_TO_GBK[3065] := 16#83A3;
   // UNICODE_TO_GBK[3066] := 16#5130;
   // UNICODE_TO_GBK[3067] := 16#83A4;
   // UNICODE_TO_GBK[3068] := 16#5131;
   // UNICODE_TO_GBK[3069] := 16#83A5;
   // UNICODE_TO_GBK[3070] := 16#5132;
   // UNICODE_TO_GBK[3071] := 16#83A6;
   // UNICODE_TO_GBK[3072] := 16#5133;
   // UNICODE_TO_GBK[3073] := 16#83A7;
   // UNICODE_TO_GBK[3074] := 16#5134;
   // UNICODE_TO_GBK[3075] := 16#83A8;
   // UNICODE_TO_GBK[3076] := 16#5135;
   // UNICODE_TO_GBK[3077] := 16#83A9;
   // UNICODE_TO_GBK[3078] := 16#5136;
   // UNICODE_TO_GBK[3079] := 16#83AA;
   // UNICODE_TO_GBK[3080] := 16#5137;
   // UNICODE_TO_GBK[3081] := 16#83AB;
   // UNICODE_TO_GBK[3082] := 16#5138;
   // UNICODE_TO_GBK[3083] := 16#83AC;
   // UNICODE_TO_GBK[3084] := 16#5139;
   // UNICODE_TO_GBK[3085] := 16#83AD;
   // UNICODE_TO_GBK[3086] := 16#513A;
   // UNICODE_TO_GBK[3087] := 16#83AE;
   // UNICODE_TO_GBK[3088] := 16#513B;
   // UNICODE_TO_GBK[3089] := 16#83AF;
   // UNICODE_TO_GBK[3090] := 16#513C;
   // UNICODE_TO_GBK[3091] := 16#83B0;
   // UNICODE_TO_GBK[3092] := 16#513D;
   // UNICODE_TO_GBK[3093] := 16#83B1;
   // UNICODE_TO_GBK[3094] := 16#513E;
   // UNICODE_TO_GBK[3095] := 16#83B2;
   // UNICODE_TO_GBK[3096] := 16#513F;
   // UNICODE_TO_GBK[3097] := 16#B6F9;
   // UNICODE_TO_GBK[3098] := 16#5140;
   // UNICODE_TO_GBK[3099] := 16#D8A3;
   // UNICODE_TO_GBK[3100] := 16#5141;
   // UNICODE_TO_GBK[3101] := 16#D4CA;
   // UNICODE_TO_GBK[3102] := 16#5142;
   // UNICODE_TO_GBK[3103] := 16#83B3;
   // UNICODE_TO_GBK[3104] := 16#5143;
   // UNICODE_TO_GBK[3105] := 16#D4AA;
   // UNICODE_TO_GBK[3106] := 16#5144;
   // UNICODE_TO_GBK[3107] := 16#D0D6;
   // UNICODE_TO_GBK[3108] := 16#5145;
   // UNICODE_TO_GBK[3109] := 16#B3E4;
   // UNICODE_TO_GBK[3110] := 16#5146;
   // UNICODE_TO_GBK[3111] := 16#D5D7;
   // UNICODE_TO_GBK[3112] := 16#5147;
   // UNICODE_TO_GBK[3113] := 16#83B4;
   // UNICODE_TO_GBK[3114] := 16#5148;
   // UNICODE_TO_GBK[3115] := 16#CFC8;
   // UNICODE_TO_GBK[3116] := 16#5149;
   // UNICODE_TO_GBK[3117] := 16#B9E2;
   // UNICODE_TO_GBK[3118] := 16#514A;
   // UNICODE_TO_GBK[3119] := 16#83B5;
   // UNICODE_TO_GBK[3120] := 16#514B;
   // UNICODE_TO_GBK[3121] := 16#BFCB;
   // UNICODE_TO_GBK[3122] := 16#514C;
   // UNICODE_TO_GBK[3123] := 16#83B6;
   // UNICODE_TO_GBK[3124] := 16#514D;
   // UNICODE_TO_GBK[3125] := 16#C3E2;
   // UNICODE_TO_GBK[3126] := 16#514E;
   // UNICODE_TO_GBK[3127] := 16#83B7;
   // UNICODE_TO_GBK[3128] := 16#514F;
   // UNICODE_TO_GBK[3129] := 16#83B8;
   // UNICODE_TO_GBK[3130] := 16#5150;
   // UNICODE_TO_GBK[3131] := 16#83B9;
   // UNICODE_TO_GBK[3132] := 16#5151;
   // UNICODE_TO_GBK[3133] := 16#B6D2;
   // UNICODE_TO_GBK[3134] := 16#5152;
   // UNICODE_TO_GBK[3135] := 16#83BA;
   // UNICODE_TO_GBK[3136] := 16#5153;
   // UNICODE_TO_GBK[3137] := 16#83BB;
   // UNICODE_TO_GBK[3138] := 16#5154;
   // UNICODE_TO_GBK[3139] := 16#CDC3;
   // UNICODE_TO_GBK[3140] := 16#5155;
   // UNICODE_TO_GBK[3141] := 16#D9EE;
   // UNICODE_TO_GBK[3142] := 16#5156;
   // UNICODE_TO_GBK[3143] := 16#D9F0;
   // UNICODE_TO_GBK[3144] := 16#5157;
   // UNICODE_TO_GBK[3145] := 16#83BC;
   // UNICODE_TO_GBK[3146] := 16#5158;
   // UNICODE_TO_GBK[3147] := 16#83BD;
   // UNICODE_TO_GBK[3148] := 16#5159;
   // UNICODE_TO_GBK[3149] := 16#83BE;
   // UNICODE_TO_GBK[3150] := 16#515A;
   // UNICODE_TO_GBK[3151] := 16#B5B3;
   // UNICODE_TO_GBK[3152] := 16#515B;
   // UNICODE_TO_GBK[3153] := 16#83BF;
   // UNICODE_TO_GBK[3154] := 16#515C;
   // UNICODE_TO_GBK[3155] := 16#B6B5;
   // UNICODE_TO_GBK[3156] := 16#515D;
   // UNICODE_TO_GBK[3157] := 16#83C0;
   // UNICODE_TO_GBK[3158] := 16#515E;
   // UNICODE_TO_GBK[3159] := 16#83C1;
   // UNICODE_TO_GBK[3160] := 16#515F;
   // UNICODE_TO_GBK[3161] := 16#83C2;
   // UNICODE_TO_GBK[3162] := 16#5160;
   // UNICODE_TO_GBK[3163] := 16#83C3;
   // UNICODE_TO_GBK[3164] := 16#5161;
   // UNICODE_TO_GBK[3165] := 16#83C4;
   // UNICODE_TO_GBK[3166] := 16#5162;
   // UNICODE_TO_GBK[3167] := 16#BEA4;
   // UNICODE_TO_GBK[3168] := 16#5163;
   // UNICODE_TO_GBK[3169] := 16#83C5;
   // UNICODE_TO_GBK[3170] := 16#5164;
   // UNICODE_TO_GBK[3171] := 16#83C6;
   // UNICODE_TO_GBK[3172] := 16#5165;
   // UNICODE_TO_GBK[3173] := 16#C8EB;
   // UNICODE_TO_GBK[3174] := 16#5166;
   // UNICODE_TO_GBK[3175] := 16#83C7;
   // UNICODE_TO_GBK[3176] := 16#5167;
   // UNICODE_TO_GBK[3177] := 16#83C8;
   // UNICODE_TO_GBK[3178] := 16#5168;
   // UNICODE_TO_GBK[3179] := 16#C8AB;
   // UNICODE_TO_GBK[3180] := 16#5169;
   // UNICODE_TO_GBK[3181] := 16#83C9;
   // UNICODE_TO_GBK[3182] := 16#516A;
   // UNICODE_TO_GBK[3183] := 16#83CA;
   // UNICODE_TO_GBK[3184] := 16#516B;
   // UNICODE_TO_GBK[3185] := 16#B0CB;
   // UNICODE_TO_GBK[3186] := 16#516C;
   // UNICODE_TO_GBK[3187] := 16#B9AB;
   // UNICODE_TO_GBK[3188] := 16#516D;
   // UNICODE_TO_GBK[3189] := 16#C1F9;
   // UNICODE_TO_GBK[3190] := 16#516E;
   // UNICODE_TO_GBK[3191] := 16#D9E2;
   // UNICODE_TO_GBK[3192] := 16#516F;
   // UNICODE_TO_GBK[3193] := 16#83CB;
   // UNICODE_TO_GBK[3194] := 16#5170;
   // UNICODE_TO_GBK[3195] := 16#C0BC;
   // UNICODE_TO_GBK[3196] := 16#5171;
   // UNICODE_TO_GBK[3197] := 16#B9B2;
   // UNICODE_TO_GBK[3198] := 16#5172;
   // UNICODE_TO_GBK[3199] := 16#83CC;
   // UNICODE_TO_GBK[3200] := 16#5173;
   // UNICODE_TO_GBK[3201] := 16#B9D8;
   // UNICODE_TO_GBK[3202] := 16#5174;
   // UNICODE_TO_GBK[3203] := 16#D0CB;
   // UNICODE_TO_GBK[3204] := 16#5175;
   // UNICODE_TO_GBK[3205] := 16#B1F8;
   // UNICODE_TO_GBK[3206] := 16#5176;
   // UNICODE_TO_GBK[3207] := 16#C6E4;
   // UNICODE_TO_GBK[3208] := 16#5177;
   // UNICODE_TO_GBK[3209] := 16#BEDF;
   // UNICODE_TO_GBK[3210] := 16#5178;
   // UNICODE_TO_GBK[3211] := 16#B5E4;
   // UNICODE_TO_GBK[3212] := 16#5179;
   // UNICODE_TO_GBK[3213] := 16#D7C8;
   // UNICODE_TO_GBK[3214] := 16#517A;
   // UNICODE_TO_GBK[3215] := 16#83CD;
   // UNICODE_TO_GBK[3216] := 16#517B;
   // UNICODE_TO_GBK[3217] := 16#D1F8;
   // UNICODE_TO_GBK[3218] := 16#517C;
   // UNICODE_TO_GBK[3219] := 16#BCE6;
   // UNICODE_TO_GBK[3220] := 16#517D;
   // UNICODE_TO_GBK[3221] := 16#CADE;
   // UNICODE_TO_GBK[3222] := 16#517E;
   // UNICODE_TO_GBK[3223] := 16#83CE;
   // UNICODE_TO_GBK[3224] := 16#517F;
   // UNICODE_TO_GBK[3225] := 16#83CF;
   // UNICODE_TO_GBK[3226] := 16#5180;
   // UNICODE_TO_GBK[3227] := 16#BCBD;
   // UNICODE_TO_GBK[3228] := 16#5181;
   // UNICODE_TO_GBK[3229] := 16#D9E6;
   // UNICODE_TO_GBK[3230] := 16#5182;
   // UNICODE_TO_GBK[3231] := 16#D8E7;
   // UNICODE_TO_GBK[3232] := 16#5183;
   // UNICODE_TO_GBK[3233] := 16#83D0;
   // UNICODE_TO_GBK[3234] := 16#5184;
   // UNICODE_TO_GBK[3235] := 16#83D1;
   // UNICODE_TO_GBK[3236] := 16#5185;
   // UNICODE_TO_GBK[3237] := 16#C4DA;
   // UNICODE_TO_GBK[3238] := 16#5186;
   // UNICODE_TO_GBK[3239] := 16#83D2;
   // UNICODE_TO_GBK[3240] := 16#5187;
   // UNICODE_TO_GBK[3241] := 16#83D3;
   // UNICODE_TO_GBK[3242] := 16#5188;
   // UNICODE_TO_GBK[3243] := 16#B8D4;
   // UNICODE_TO_GBK[3244] := 16#5189;
   // UNICODE_TO_GBK[3245] := 16#C8BD;
   // UNICODE_TO_GBK[3246] := 16#518A;
   // UNICODE_TO_GBK[3247] := 16#83D4;
   // UNICODE_TO_GBK[3248] := 16#518B;
   // UNICODE_TO_GBK[3249] := 16#83D5;
   // UNICODE_TO_GBK[3250] := 16#518C;
   // UNICODE_TO_GBK[3251] := 16#B2E1;
   // UNICODE_TO_GBK[3252] := 16#518D;
   // UNICODE_TO_GBK[3253] := 16#D4D9;
   // UNICODE_TO_GBK[3254] := 16#518E;
   // UNICODE_TO_GBK[3255] := 16#83D6;
   // UNICODE_TO_GBK[3256] := 16#518F;
   // UNICODE_TO_GBK[3257] := 16#83D7;
   // UNICODE_TO_GBK[3258] := 16#5190;
   // UNICODE_TO_GBK[3259] := 16#83D8;
   // UNICODE_TO_GBK[3260] := 16#5191;
   // UNICODE_TO_GBK[3261] := 16#83D9;
   // UNICODE_TO_GBK[3262] := 16#5192;
   // UNICODE_TO_GBK[3263] := 16#C3B0;
   // UNICODE_TO_GBK[3264] := 16#5193;
   // UNICODE_TO_GBK[3265] := 16#83DA;
   // UNICODE_TO_GBK[3266] := 16#5194;
   // UNICODE_TO_GBK[3267] := 16#83DB;
   // UNICODE_TO_GBK[3268] := 16#5195;
   // UNICODE_TO_GBK[3269] := 16#C3E1;
   // UNICODE_TO_GBK[3270] := 16#5196;
   // UNICODE_TO_GBK[3271] := 16#DAA2;
   // UNICODE_TO_GBK[3272] := 16#5197;
   // UNICODE_TO_GBK[3273] := 16#C8DF;
   // UNICODE_TO_GBK[3274] := 16#5198;
   // UNICODE_TO_GBK[3275] := 16#83DC;
   // UNICODE_TO_GBK[3276] := 16#5199;
   // UNICODE_TO_GBK[3277] := 16#D0B4;
   // UNICODE_TO_GBK[3278] := 16#519A;
   // UNICODE_TO_GBK[3279] := 16#83DD;
   // UNICODE_TO_GBK[3280] := 16#519B;
   // UNICODE_TO_GBK[3281] := 16#BEFC;
   // UNICODE_TO_GBK[3282] := 16#519C;
   // UNICODE_TO_GBK[3283] := 16#C5A9;
   // UNICODE_TO_GBK[3284] := 16#519D;
   // UNICODE_TO_GBK[3285] := 16#83DE;
   // UNICODE_TO_GBK[3286] := 16#519E;
   // UNICODE_TO_GBK[3287] := 16#83DF;
   // UNICODE_TO_GBK[3288] := 16#519F;
   // UNICODE_TO_GBK[3289] := 16#83E0;
   // UNICODE_TO_GBK[3290] := 16#51A0;
   // UNICODE_TO_GBK[3291] := 16#B9DA;
   // UNICODE_TO_GBK[3292] := 16#51A1;
   // UNICODE_TO_GBK[3293] := 16#83E1;
   // UNICODE_TO_GBK[3294] := 16#51A2;
   // UNICODE_TO_GBK[3295] := 16#DAA3;
   // UNICODE_TO_GBK[3296] := 16#51A3;
   // UNICODE_TO_GBK[3297] := 16#83E2;
   // UNICODE_TO_GBK[3298] := 16#51A4;
   // UNICODE_TO_GBK[3299] := 16#D4A9;
   // UNICODE_TO_GBK[3300] := 16#51A5;
   // UNICODE_TO_GBK[3301] := 16#DAA4;
   // UNICODE_TO_GBK[3302] := 16#51A6;
   // UNICODE_TO_GBK[3303] := 16#83E3;
   // UNICODE_TO_GBK[3304] := 16#51A7;
   // UNICODE_TO_GBK[3305] := 16#83E4;
   // UNICODE_TO_GBK[3306] := 16#51A8;
   // UNICODE_TO_GBK[3307] := 16#83E5;
   // UNICODE_TO_GBK[3308] := 16#51A9;
   // UNICODE_TO_GBK[3309] := 16#83E6;
   // UNICODE_TO_GBK[3310] := 16#51AA;
   // UNICODE_TO_GBK[3311] := 16#83E7;
   // UNICODE_TO_GBK[3312] := 16#51AB;
   // UNICODE_TO_GBK[3313] := 16#D9FB;
   // UNICODE_TO_GBK[3314] := 16#51AC;
   // UNICODE_TO_GBK[3315] := 16#B6AC;
   // UNICODE_TO_GBK[3316] := 16#51AD;
   // UNICODE_TO_GBK[3317] := 16#83E8;
   // UNICODE_TO_GBK[3318] := 16#51AE;
   // UNICODE_TO_GBK[3319] := 16#83E9;
   // UNICODE_TO_GBK[3320] := 16#51AF;
   // UNICODE_TO_GBK[3321] := 16#B7EB;
   // UNICODE_TO_GBK[3322] := 16#51B0;
   // UNICODE_TO_GBK[3323] := 16#B1F9;
   // UNICODE_TO_GBK[3324] := 16#51B1;
   // UNICODE_TO_GBK[3325] := 16#D9FC;
   // UNICODE_TO_GBK[3326] := 16#51B2;
   // UNICODE_TO_GBK[3327] := 16#B3E5;
   // UNICODE_TO_GBK[3328] := 16#51B3;
   // UNICODE_TO_GBK[3329] := 16#BEF6;
   // UNICODE_TO_GBK[3330] := 16#51B4;
   // UNICODE_TO_GBK[3331] := 16#83EA;
   // UNICODE_TO_GBK[3332] := 16#51B5;
   // UNICODE_TO_GBK[3333] := 16#BFF6;
   // UNICODE_TO_GBK[3334] := 16#51B6;
   // UNICODE_TO_GBK[3335] := 16#D2B1;
   // UNICODE_TO_GBK[3336] := 16#51B7;
   // UNICODE_TO_GBK[3337] := 16#C0E4;
   // UNICODE_TO_GBK[3338] := 16#51B8;
   // UNICODE_TO_GBK[3339] := 16#83EB;
   // UNICODE_TO_GBK[3340] := 16#51B9;
   // UNICODE_TO_GBK[3341] := 16#83EC;
   // UNICODE_TO_GBK[3342] := 16#51BA;
   // UNICODE_TO_GBK[3343] := 16#83ED;
   // UNICODE_TO_GBK[3344] := 16#51BB;
   // UNICODE_TO_GBK[3345] := 16#B6B3;
   // UNICODE_TO_GBK[3346] := 16#51BC;
   // UNICODE_TO_GBK[3347] := 16#D9FE;
   // UNICODE_TO_GBK[3348] := 16#51BD;
   // UNICODE_TO_GBK[3349] := 16#D9FD;
   // UNICODE_TO_GBK[3350] := 16#51BE;
   // UNICODE_TO_GBK[3351] := 16#83EE;
   // UNICODE_TO_GBK[3352] := 16#51BF;
   // UNICODE_TO_GBK[3353] := 16#83EF;
   // UNICODE_TO_GBK[3354] := 16#51C0;
   // UNICODE_TO_GBK[3355] := 16#BEBB;
   // UNICODE_TO_GBK[3356] := 16#51C1;
   // UNICODE_TO_GBK[3357] := 16#83F0;
   // UNICODE_TO_GBK[3358] := 16#51C2;
   // UNICODE_TO_GBK[3359] := 16#83F1;
   // UNICODE_TO_GBK[3360] := 16#51C3;
   // UNICODE_TO_GBK[3361] := 16#83F2;
   // UNICODE_TO_GBK[3362] := 16#51C4;
   // UNICODE_TO_GBK[3363] := 16#C6E0;
   // UNICODE_TO_GBK[3364] := 16#51C5;
   // UNICODE_TO_GBK[3365] := 16#83F3;
   // UNICODE_TO_GBK[3366] := 16#51C6;
   // UNICODE_TO_GBK[3367] := 16#D7BC;
   // UNICODE_TO_GBK[3368] := 16#51C7;
   // UNICODE_TO_GBK[3369] := 16#DAA1;
   // UNICODE_TO_GBK[3370] := 16#51C8;
   // UNICODE_TO_GBK[3371] := 16#83F4;
   // UNICODE_TO_GBK[3372] := 16#51C9;
   // UNICODE_TO_GBK[3373] := 16#C1B9;
   // UNICODE_TO_GBK[3374] := 16#51CA;
   // UNICODE_TO_GBK[3375] := 16#83F5;
   // UNICODE_TO_GBK[3376] := 16#51CB;
   // UNICODE_TO_GBK[3377] := 16#B5F2;
   // UNICODE_TO_GBK[3378] := 16#51CC;
   // UNICODE_TO_GBK[3379] := 16#C1E8;
   // UNICODE_TO_GBK[3380] := 16#51CD;
   // UNICODE_TO_GBK[3381] := 16#83F6;
   // UNICODE_TO_GBK[3382] := 16#51CE;
   // UNICODE_TO_GBK[3383] := 16#83F7;
   // UNICODE_TO_GBK[3384] := 16#51CF;
   // UNICODE_TO_GBK[3385] := 16#BCF5;
   // UNICODE_TO_GBK[3386] := 16#51D0;
   // UNICODE_TO_GBK[3387] := 16#83F8;
   // UNICODE_TO_GBK[3388] := 16#51D1;
   // UNICODE_TO_GBK[3389] := 16#B4D5;
   // UNICODE_TO_GBK[3390] := 16#51D2;
   // UNICODE_TO_GBK[3391] := 16#83F9;
   // UNICODE_TO_GBK[3392] := 16#51D3;
   // UNICODE_TO_GBK[3393] := 16#83FA;
   // UNICODE_TO_GBK[3394] := 16#51D4;
   // UNICODE_TO_GBK[3395] := 16#83FB;
   // UNICODE_TO_GBK[3396] := 16#51D5;
   // UNICODE_TO_GBK[3397] := 16#83FC;
   // UNICODE_TO_GBK[3398] := 16#51D6;
   // UNICODE_TO_GBK[3399] := 16#83FD;
   // UNICODE_TO_GBK[3400] := 16#51D7;
   // UNICODE_TO_GBK[3401] := 16#83FE;
   // UNICODE_TO_GBK[3402] := 16#51D8;
   // UNICODE_TO_GBK[3403] := 16#8440;
   // UNICODE_TO_GBK[3404] := 16#51D9;
   // UNICODE_TO_GBK[3405] := 16#8441;
   // UNICODE_TO_GBK[3406] := 16#51DA;
   // UNICODE_TO_GBK[3407] := 16#8442;
   // UNICODE_TO_GBK[3408] := 16#51DB;
   // UNICODE_TO_GBK[3409] := 16#C1DD;
   // UNICODE_TO_GBK[3410] := 16#51DC;
   // UNICODE_TO_GBK[3411] := 16#8443;
   // UNICODE_TO_GBK[3412] := 16#51DD;
   // UNICODE_TO_GBK[3413] := 16#C4FD;
   // UNICODE_TO_GBK[3414] := 16#51DE;
   // UNICODE_TO_GBK[3415] := 16#8444;
   // UNICODE_TO_GBK[3416] := 16#51DF;
   // UNICODE_TO_GBK[3417] := 16#8445;
   // UNICODE_TO_GBK[3418] := 16#51E0;
   // UNICODE_TO_GBK[3419] := 16#BCB8;
   // UNICODE_TO_GBK[3420] := 16#51E1;
   // UNICODE_TO_GBK[3421] := 16#B7B2;
   // UNICODE_TO_GBK[3422] := 16#51E2;
   // UNICODE_TO_GBK[3423] := 16#8446;
   // UNICODE_TO_GBK[3424] := 16#51E3;
   // UNICODE_TO_GBK[3425] := 16#8447;
   // UNICODE_TO_GBK[3426] := 16#51E4;
   // UNICODE_TO_GBK[3427] := 16#B7EF;
   // UNICODE_TO_GBK[3428] := 16#51E5;
   // UNICODE_TO_GBK[3429] := 16#8448;
   // UNICODE_TO_GBK[3430] := 16#51E6;
   // UNICODE_TO_GBK[3431] := 16#8449;
   // UNICODE_TO_GBK[3432] := 16#51E7;
   // UNICODE_TO_GBK[3433] := 16#844A;
   // UNICODE_TO_GBK[3434] := 16#51E8;
   // UNICODE_TO_GBK[3435] := 16#844B;
   // UNICODE_TO_GBK[3436] := 16#51E9;
   // UNICODE_TO_GBK[3437] := 16#844C;
   // UNICODE_TO_GBK[3438] := 16#51EA;
   // UNICODE_TO_GBK[3439] := 16#844D;
   // UNICODE_TO_GBK[3440] := 16#51EB;
   // UNICODE_TO_GBK[3441] := 16#D9EC;
   // UNICODE_TO_GBK[3442] := 16#51EC;
   // UNICODE_TO_GBK[3443] := 16#844E;
   // UNICODE_TO_GBK[3444] := 16#51ED;
   // UNICODE_TO_GBK[3445] := 16#C6BE;
   // UNICODE_TO_GBK[3446] := 16#51EE;
   // UNICODE_TO_GBK[3447] := 16#844F;
   // UNICODE_TO_GBK[3448] := 16#51EF;
   // UNICODE_TO_GBK[3449] := 16#BFAD;
   // UNICODE_TO_GBK[3450] := 16#51F0;
   // UNICODE_TO_GBK[3451] := 16#BBCB;
   // UNICODE_TO_GBK[3452] := 16#51F1;
   // UNICODE_TO_GBK[3453] := 16#8450;
   // UNICODE_TO_GBK[3454] := 16#51F2;
   // UNICODE_TO_GBK[3455] := 16#8451;
   // UNICODE_TO_GBK[3456] := 16#51F3;
   // UNICODE_TO_GBK[3457] := 16#B5CA;
   // UNICODE_TO_GBK[3458] := 16#51F4;
   // UNICODE_TO_GBK[3459] := 16#8452;
   // UNICODE_TO_GBK[3460] := 16#51F5;
   // UNICODE_TO_GBK[3461] := 16#DBC9;
   // UNICODE_TO_GBK[3462] := 16#51F6;
   // UNICODE_TO_GBK[3463] := 16#D0D7;
   // UNICODE_TO_GBK[3464] := 16#51F7;
   // UNICODE_TO_GBK[3465] := 16#8453;
   // UNICODE_TO_GBK[3466] := 16#51F8;
   // UNICODE_TO_GBK[3467] := 16#CDB9;
   // UNICODE_TO_GBK[3468] := 16#51F9;
   // UNICODE_TO_GBK[3469] := 16#B0BC;
   // UNICODE_TO_GBK[3470] := 16#51FA;
   // UNICODE_TO_GBK[3471] := 16#B3F6;
   // UNICODE_TO_GBK[3472] := 16#51FB;
   // UNICODE_TO_GBK[3473] := 16#BBF7;
   // UNICODE_TO_GBK[3474] := 16#51FC;
   // UNICODE_TO_GBK[3475] := 16#DBCA;
   // UNICODE_TO_GBK[3476] := 16#51FD;
   // UNICODE_TO_GBK[3477] := 16#BAAF;
   // UNICODE_TO_GBK[3478] := 16#51FE;
   // UNICODE_TO_GBK[3479] := 16#8454;
   // UNICODE_TO_GBK[3480] := 16#51FF;
   // UNICODE_TO_GBK[3481] := 16#D4E4;
   // UNICODE_TO_GBK[3482] := 16#5200;
   // UNICODE_TO_GBK[3483] := 16#B5B6;
   // UNICODE_TO_GBK[3484] := 16#5201;
   // UNICODE_TO_GBK[3485] := 16#B5F3;
   // UNICODE_TO_GBK[3486] := 16#5202;
   // UNICODE_TO_GBK[3487] := 16#D8D6;
   // UNICODE_TO_GBK[3488] := 16#5203;
   // UNICODE_TO_GBK[3489] := 16#C8D0;
   // UNICODE_TO_GBK[3490] := 16#5204;
   // UNICODE_TO_GBK[3491] := 16#8455;
   // UNICODE_TO_GBK[3492] := 16#5205;
   // UNICODE_TO_GBK[3493] := 16#8456;
   // UNICODE_TO_GBK[3494] := 16#5206;
   // UNICODE_TO_GBK[3495] := 16#B7D6;
   // UNICODE_TO_GBK[3496] := 16#5207;
   // UNICODE_TO_GBK[3497] := 16#C7D0;
   // UNICODE_TO_GBK[3498] := 16#5208;
   // UNICODE_TO_GBK[3499] := 16#D8D7;
   // UNICODE_TO_GBK[3500] := 16#5209;
   // UNICODE_TO_GBK[3501] := 16#8457;
   // UNICODE_TO_GBK[3502] := 16#520A;
   // UNICODE_TO_GBK[3503] := 16#BFAF;
   // UNICODE_TO_GBK[3504] := 16#520B;
   // UNICODE_TO_GBK[3505] := 16#8458;
   // UNICODE_TO_GBK[3506] := 16#520C;
   // UNICODE_TO_GBK[3507] := 16#8459;
   // UNICODE_TO_GBK[3508] := 16#520D;
   // UNICODE_TO_GBK[3509] := 16#DBBB;
   // UNICODE_TO_GBK[3510] := 16#520E;
   // UNICODE_TO_GBK[3511] := 16#D8D8;
   // UNICODE_TO_GBK[3512] := 16#520F;
   // UNICODE_TO_GBK[3513] := 16#845A;
   // UNICODE_TO_GBK[3514] := 16#5210;
   // UNICODE_TO_GBK[3515] := 16#845B;
   // UNICODE_TO_GBK[3516] := 16#5211;
   // UNICODE_TO_GBK[3517] := 16#D0CC;
   // UNICODE_TO_GBK[3518] := 16#5212;
   // UNICODE_TO_GBK[3519] := 16#BBAE;
   // UNICODE_TO_GBK[3520] := 16#5213;
   // UNICODE_TO_GBK[3521] := 16#845C;
   // UNICODE_TO_GBK[3522] := 16#5214;
   // UNICODE_TO_GBK[3523] := 16#845D;
   // UNICODE_TO_GBK[3524] := 16#5215;
   // UNICODE_TO_GBK[3525] := 16#845E;
   // UNICODE_TO_GBK[3526] := 16#5216;
   // UNICODE_TO_GBK[3527] := 16#EBBE;
   // UNICODE_TO_GBK[3528] := 16#5217;
   // UNICODE_TO_GBK[3529] := 16#C1D0;
   // UNICODE_TO_GBK[3530] := 16#5218;
   // UNICODE_TO_GBK[3531] := 16#C1F5;
   // UNICODE_TO_GBK[3532] := 16#5219;
   // UNICODE_TO_GBK[3533] := 16#D4F2;
   // UNICODE_TO_GBK[3534] := 16#521A;
   // UNICODE_TO_GBK[3535] := 16#B8D5;
   // UNICODE_TO_GBK[3536] := 16#521B;
   // UNICODE_TO_GBK[3537] := 16#B4B4;
   // UNICODE_TO_GBK[3538] := 16#521C;
   // UNICODE_TO_GBK[3539] := 16#845F;
   // UNICODE_TO_GBK[3540] := 16#521D;
   // UNICODE_TO_GBK[3541] := 16#B3F5;
   // UNICODE_TO_GBK[3542] := 16#521E;
   // UNICODE_TO_GBK[3543] := 16#8460;
   // UNICODE_TO_GBK[3544] := 16#521F;
   // UNICODE_TO_GBK[3545] := 16#8461;
   // UNICODE_TO_GBK[3546] := 16#5220;
   // UNICODE_TO_GBK[3547] := 16#C9BE;
   // UNICODE_TO_GBK[3548] := 16#5221;
   // UNICODE_TO_GBK[3549] := 16#8462;
   // UNICODE_TO_GBK[3550] := 16#5222;
   // UNICODE_TO_GBK[3551] := 16#8463;
   // UNICODE_TO_GBK[3552] := 16#5223;
   // UNICODE_TO_GBK[3553] := 16#8464;
   // UNICODE_TO_GBK[3554] := 16#5224;
   // UNICODE_TO_GBK[3555] := 16#C5D0;
   // UNICODE_TO_GBK[3556] := 16#5225;
   // UNICODE_TO_GBK[3557] := 16#8465;
   // UNICODE_TO_GBK[3558] := 16#5226;
   // UNICODE_TO_GBK[3559] := 16#8466;
   // UNICODE_TO_GBK[3560] := 16#5227;
   // UNICODE_TO_GBK[3561] := 16#8467;
   // UNICODE_TO_GBK[3562] := 16#5228;
   // UNICODE_TO_GBK[3563] := 16#C5D9;
   // UNICODE_TO_GBK[3564] := 16#5229;
   // UNICODE_TO_GBK[3565] := 16#C0FB;
   // UNICODE_TO_GBK[3566] := 16#522A;
   // UNICODE_TO_GBK[3567] := 16#8468;
   // UNICODE_TO_GBK[3568] := 16#522B;
   // UNICODE_TO_GBK[3569] := 16#B1F0;
   // UNICODE_TO_GBK[3570] := 16#522C;
   // UNICODE_TO_GBK[3571] := 16#8469;
   // UNICODE_TO_GBK[3572] := 16#522D;
   // UNICODE_TO_GBK[3573] := 16#D8D9;
   // UNICODE_TO_GBK[3574] := 16#522E;
   // UNICODE_TO_GBK[3575] := 16#B9CE;
   // UNICODE_TO_GBK[3576] := 16#522F;
   // UNICODE_TO_GBK[3577] := 16#846A;
   // UNICODE_TO_GBK[3578] := 16#5230;
   // UNICODE_TO_GBK[3579] := 16#B5BD;
   // UNICODE_TO_GBK[3580] := 16#5231;
   // UNICODE_TO_GBK[3581] := 16#846B;
   // UNICODE_TO_GBK[3582] := 16#5232;
   // UNICODE_TO_GBK[3583] := 16#846C;
   // UNICODE_TO_GBK[3584] := 16#5233;
   // UNICODE_TO_GBK[3585] := 16#D8DA;
   // UNICODE_TO_GBK[3586] := 16#5234;
   // UNICODE_TO_GBK[3587] := 16#846D;
   // UNICODE_TO_GBK[3588] := 16#5235;
   // UNICODE_TO_GBK[3589] := 16#846E;
   // UNICODE_TO_GBK[3590] := 16#5236;
   // UNICODE_TO_GBK[3591] := 16#D6C6;
   // UNICODE_TO_GBK[3592] := 16#5237;
   // UNICODE_TO_GBK[3593] := 16#CBA2;
   // UNICODE_TO_GBK[3594] := 16#5238;
   // UNICODE_TO_GBK[3595] := 16#C8AF;
   // UNICODE_TO_GBK[3596] := 16#5239;
   // UNICODE_TO_GBK[3597] := 16#C9B2;
   // UNICODE_TO_GBK[3598] := 16#523A;
   // UNICODE_TO_GBK[3599] := 16#B4CC;
   // UNICODE_TO_GBK[3600] := 16#523B;
   // UNICODE_TO_GBK[3601] := 16#BFCC;
   // UNICODE_TO_GBK[3602] := 16#523C;
   // UNICODE_TO_GBK[3603] := 16#846F;
   // UNICODE_TO_GBK[3604] := 16#523D;
   // UNICODE_TO_GBK[3605] := 16#B9F4;
   // UNICODE_TO_GBK[3606] := 16#523E;
   // UNICODE_TO_GBK[3607] := 16#8470;
   // UNICODE_TO_GBK[3608] := 16#523F;
   // UNICODE_TO_GBK[3609] := 16#D8DB;
   // UNICODE_TO_GBK[3610] := 16#5240;
   // UNICODE_TO_GBK[3611] := 16#D8DC;
   // UNICODE_TO_GBK[3612] := 16#5241;
   // UNICODE_TO_GBK[3613] := 16#B6E7;
   // UNICODE_TO_GBK[3614] := 16#5242;
   // UNICODE_TO_GBK[3615] := 16#BCC1;
   // UNICODE_TO_GBK[3616] := 16#5243;
   // UNICODE_TO_GBK[3617] := 16#CCEA;
   // UNICODE_TO_GBK[3618] := 16#5244;
   // UNICODE_TO_GBK[3619] := 16#8471;
   // UNICODE_TO_GBK[3620] := 16#5245;
   // UNICODE_TO_GBK[3621] := 16#8472;
   // UNICODE_TO_GBK[3622] := 16#5246;
   // UNICODE_TO_GBK[3623] := 16#8473;
   // UNICODE_TO_GBK[3624] := 16#5247;
   // UNICODE_TO_GBK[3625] := 16#8474;
   // UNICODE_TO_GBK[3626] := 16#5248;
   // UNICODE_TO_GBK[3627] := 16#8475;
   // UNICODE_TO_GBK[3628] := 16#5249;
   // UNICODE_TO_GBK[3629] := 16#8476;
   // UNICODE_TO_GBK[3630] := 16#524A;
   // UNICODE_TO_GBK[3631] := 16#CFF7;
   // UNICODE_TO_GBK[3632] := 16#524B;
   // UNICODE_TO_GBK[3633] := 16#8477;
   // UNICODE_TO_GBK[3634] := 16#524C;
   // UNICODE_TO_GBK[3635] := 16#D8DD;
   // UNICODE_TO_GBK[3636] := 16#524D;
   // UNICODE_TO_GBK[3637] := 16#C7B0;
   // UNICODE_TO_GBK[3638] := 16#524E;
   // UNICODE_TO_GBK[3639] := 16#8478;
   // UNICODE_TO_GBK[3640] := 16#524F;
   // UNICODE_TO_GBK[3641] := 16#8479;
   // UNICODE_TO_GBK[3642] := 16#5250;
   // UNICODE_TO_GBK[3643] := 16#B9D0;
   // UNICODE_TO_GBK[3644] := 16#5251;
   // UNICODE_TO_GBK[3645] := 16#BDA3;
   // UNICODE_TO_GBK[3646] := 16#5252;
   // UNICODE_TO_GBK[3647] := 16#847A;
   // UNICODE_TO_GBK[3648] := 16#5253;
   // UNICODE_TO_GBK[3649] := 16#847B;
   // UNICODE_TO_GBK[3650] := 16#5254;
   // UNICODE_TO_GBK[3651] := 16#CCDE;
   // UNICODE_TO_GBK[3652] := 16#5255;
   // UNICODE_TO_GBK[3653] := 16#847C;
   // UNICODE_TO_GBK[3654] := 16#5256;
   // UNICODE_TO_GBK[3655] := 16#C6CA;
   // UNICODE_TO_GBK[3656] := 16#5257;
   // UNICODE_TO_GBK[3657] := 16#847D;
   // UNICODE_TO_GBK[3658] := 16#5258;
   // UNICODE_TO_GBK[3659] := 16#847E;
   // UNICODE_TO_GBK[3660] := 16#5259;
   // UNICODE_TO_GBK[3661] := 16#8480;
   // UNICODE_TO_GBK[3662] := 16#525A;
   // UNICODE_TO_GBK[3663] := 16#8481;
   // UNICODE_TO_GBK[3664] := 16#525B;
   // UNICODE_TO_GBK[3665] := 16#8482;
   // UNICODE_TO_GBK[3666] := 16#525C;
   // UNICODE_TO_GBK[3667] := 16#D8E0;
   // UNICODE_TO_GBK[3668] := 16#525D;
   // UNICODE_TO_GBK[3669] := 16#8483;
   // UNICODE_TO_GBK[3670] := 16#525E;
   // UNICODE_TO_GBK[3671] := 16#D8DE;
   // UNICODE_TO_GBK[3672] := 16#525F;
   // UNICODE_TO_GBK[3673] := 16#8484;
   // UNICODE_TO_GBK[3674] := 16#5260;
   // UNICODE_TO_GBK[3675] := 16#8485;
   // UNICODE_TO_GBK[3676] := 16#5261;
   // UNICODE_TO_GBK[3677] := 16#D8DF;
   // UNICODE_TO_GBK[3678] := 16#5262;
   // UNICODE_TO_GBK[3679] := 16#8486;
   // UNICODE_TO_GBK[3680] := 16#5263;
   // UNICODE_TO_GBK[3681] := 16#8487;
   // UNICODE_TO_GBK[3682] := 16#5264;
   // UNICODE_TO_GBK[3683] := 16#8488;
   // UNICODE_TO_GBK[3684] := 16#5265;
   // UNICODE_TO_GBK[3685] := 16#B0FE;
   // UNICODE_TO_GBK[3686] := 16#5266;
   // UNICODE_TO_GBK[3687] := 16#8489;
   // UNICODE_TO_GBK[3688] := 16#5267;
   // UNICODE_TO_GBK[3689] := 16#BEE7;
   // UNICODE_TO_GBK[3690] := 16#5268;
   // UNICODE_TO_GBK[3691] := 16#848A;
   // UNICODE_TO_GBK[3692] := 16#5269;
   // UNICODE_TO_GBK[3693] := 16#CAA3;
   // UNICODE_TO_GBK[3694] := 16#526A;
   // UNICODE_TO_GBK[3695] := 16#BCF4;
   // UNICODE_TO_GBK[3696] := 16#526B;
   // UNICODE_TO_GBK[3697] := 16#848B;
   // UNICODE_TO_GBK[3698] := 16#526C;
   // UNICODE_TO_GBK[3699] := 16#848C;
   // UNICODE_TO_GBK[3700] := 16#526D;
   // UNICODE_TO_GBK[3701] := 16#848D;
   // UNICODE_TO_GBK[3702] := 16#526E;
   // UNICODE_TO_GBK[3703] := 16#848E;
   // UNICODE_TO_GBK[3704] := 16#526F;
   // UNICODE_TO_GBK[3705] := 16#B8B1;
   // UNICODE_TO_GBK[3706] := 16#5270;
   // UNICODE_TO_GBK[3707] := 16#848F;
   // UNICODE_TO_GBK[3708] := 16#5271;
   // UNICODE_TO_GBK[3709] := 16#8490;
   // UNICODE_TO_GBK[3710] := 16#5272;
   // UNICODE_TO_GBK[3711] := 16#B8EE;
   // UNICODE_TO_GBK[3712] := 16#5273;
   // UNICODE_TO_GBK[3713] := 16#8491;
   // UNICODE_TO_GBK[3714] := 16#5274;
   // UNICODE_TO_GBK[3715] := 16#8492;
   // UNICODE_TO_GBK[3716] := 16#5275;
   // UNICODE_TO_GBK[3717] := 16#8493;
   // UNICODE_TO_GBK[3718] := 16#5276;
   // UNICODE_TO_GBK[3719] := 16#8494;
   // UNICODE_TO_GBK[3720] := 16#5277;
   // UNICODE_TO_GBK[3721] := 16#8495;
   // UNICODE_TO_GBK[3722] := 16#5278;
   // UNICODE_TO_GBK[3723] := 16#8496;
   // UNICODE_TO_GBK[3724] := 16#5279;
   // UNICODE_TO_GBK[3725] := 16#8497;
   // UNICODE_TO_GBK[3726] := 16#527A;
   // UNICODE_TO_GBK[3727] := 16#8498;
   // UNICODE_TO_GBK[3728] := 16#527B;
   // UNICODE_TO_GBK[3729] := 16#8499;
   // UNICODE_TO_GBK[3730] := 16#527C;
   // UNICODE_TO_GBK[3731] := 16#849A;
   // UNICODE_TO_GBK[3732] := 16#527D;
   // UNICODE_TO_GBK[3733] := 16#D8E2;
   // UNICODE_TO_GBK[3734] := 16#527E;
   // UNICODE_TO_GBK[3735] := 16#849B;
   // UNICODE_TO_GBK[3736] := 16#527F;
   // UNICODE_TO_GBK[3737] := 16#BDCB;
   // UNICODE_TO_GBK[3738] := 16#5280;
   // UNICODE_TO_GBK[3739] := 16#849C;
   // UNICODE_TO_GBK[3740] := 16#5281;
   // UNICODE_TO_GBK[3741] := 16#D8E4;
   // UNICODE_TO_GBK[3742] := 16#5282;
   // UNICODE_TO_GBK[3743] := 16#D8E3;
   // UNICODE_TO_GBK[3744] := 16#5283;
   // UNICODE_TO_GBK[3745] := 16#849D;
   // UNICODE_TO_GBK[3746] := 16#5284;
   // UNICODE_TO_GBK[3747] := 16#849E;
   // UNICODE_TO_GBK[3748] := 16#5285;
   // UNICODE_TO_GBK[3749] := 16#849F;
   // UNICODE_TO_GBK[3750] := 16#5286;
   // UNICODE_TO_GBK[3751] := 16#84A0;
   // UNICODE_TO_GBK[3752] := 16#5287;
   // UNICODE_TO_GBK[3753] := 16#84A1;
   // UNICODE_TO_GBK[3754] := 16#5288;
   // UNICODE_TO_GBK[3755] := 16#C5FC;
   // UNICODE_TO_GBK[3756] := 16#5289;
   // UNICODE_TO_GBK[3757] := 16#84A2;
   // UNICODE_TO_GBK[3758] := 16#528A;
   // UNICODE_TO_GBK[3759] := 16#84A3;
   // UNICODE_TO_GBK[3760] := 16#528B;
   // UNICODE_TO_GBK[3761] := 16#84A4;
   // UNICODE_TO_GBK[3762] := 16#528C;
   // UNICODE_TO_GBK[3763] := 16#84A5;
   // UNICODE_TO_GBK[3764] := 16#528D;
   // UNICODE_TO_GBK[3765] := 16#84A6;
   // UNICODE_TO_GBK[3766] := 16#528E;
   // UNICODE_TO_GBK[3767] := 16#84A7;
   // UNICODE_TO_GBK[3768] := 16#528F;
   // UNICODE_TO_GBK[3769] := 16#84A8;
   // UNICODE_TO_GBK[3770] := 16#5290;
   // UNICODE_TO_GBK[3771] := 16#D8E5;
   // UNICODE_TO_GBK[3772] := 16#5291;
   // UNICODE_TO_GBK[3773] := 16#84A9;
   // UNICODE_TO_GBK[3774] := 16#5292;
   // UNICODE_TO_GBK[3775] := 16#84AA;
   // UNICODE_TO_GBK[3776] := 16#5293;
   // UNICODE_TO_GBK[3777] := 16#D8E6;
   // UNICODE_TO_GBK[3778] := 16#5294;
   // UNICODE_TO_GBK[3779] := 16#84AB;
   // UNICODE_TO_GBK[3780] := 16#5295;
   // UNICODE_TO_GBK[3781] := 16#84AC;
   // UNICODE_TO_GBK[3782] := 16#5296;
   // UNICODE_TO_GBK[3783] := 16#84AD;
   // UNICODE_TO_GBK[3784] := 16#5297;
   // UNICODE_TO_GBK[3785] := 16#84AE;
   // UNICODE_TO_GBK[3786] := 16#5298;
   // UNICODE_TO_GBK[3787] := 16#84AF;
   // UNICODE_TO_GBK[3788] := 16#5299;
   // UNICODE_TO_GBK[3789] := 16#84B0;
   // UNICODE_TO_GBK[3790] := 16#529A;
   // UNICODE_TO_GBK[3791] := 16#84B1;
   // UNICODE_TO_GBK[3792] := 16#529B;
   // UNICODE_TO_GBK[3793] := 16#C1A6;
   // UNICODE_TO_GBK[3794] := 16#529C;
   // UNICODE_TO_GBK[3795] := 16#84B2;
   // UNICODE_TO_GBK[3796] := 16#529D;
   // UNICODE_TO_GBK[3797] := 16#C8B0;
   // UNICODE_TO_GBK[3798] := 16#529E;
   // UNICODE_TO_GBK[3799] := 16#B0EC;
   // UNICODE_TO_GBK[3800] := 16#529F;
   // UNICODE_TO_GBK[3801] := 16#B9A6;
   // UNICODE_TO_GBK[3802] := 16#52A0;
   // UNICODE_TO_GBK[3803] := 16#BCD3;
   // UNICODE_TO_GBK[3804] := 16#52A1;
   // UNICODE_TO_GBK[3805] := 16#CEF1;
   // UNICODE_TO_GBK[3806] := 16#52A2;
   // UNICODE_TO_GBK[3807] := 16#DBBD;
   // UNICODE_TO_GBK[3808] := 16#52A3;
   // UNICODE_TO_GBK[3809] := 16#C1D3;
   // UNICODE_TO_GBK[3810] := 16#52A4;
   // UNICODE_TO_GBK[3811] := 16#84B3;
   // UNICODE_TO_GBK[3812] := 16#52A5;
   // UNICODE_TO_GBK[3813] := 16#84B4;
   // UNICODE_TO_GBK[3814] := 16#52A6;
   // UNICODE_TO_GBK[3815] := 16#84B5;
   // UNICODE_TO_GBK[3816] := 16#52A7;
   // UNICODE_TO_GBK[3817] := 16#84B6;
   // UNICODE_TO_GBK[3818] := 16#52A8;
   // UNICODE_TO_GBK[3819] := 16#B6AF;
   // UNICODE_TO_GBK[3820] := 16#52A9;
   // UNICODE_TO_GBK[3821] := 16#D6FA;
   // UNICODE_TO_GBK[3822] := 16#52AA;
   // UNICODE_TO_GBK[3823] := 16#C5AC;
   // UNICODE_TO_GBK[3824] := 16#52AB;
   // UNICODE_TO_GBK[3825] := 16#BDD9;
   // UNICODE_TO_GBK[3826] := 16#52AC;
   // UNICODE_TO_GBK[3827] := 16#DBBE;
   // UNICODE_TO_GBK[3828] := 16#52AD;
   // UNICODE_TO_GBK[3829] := 16#DBBF;
   // UNICODE_TO_GBK[3830] := 16#52AE;
   // UNICODE_TO_GBK[3831] := 16#84B7;
   // UNICODE_TO_GBK[3832] := 16#52AF;
   // UNICODE_TO_GBK[3833] := 16#84B8;
   // UNICODE_TO_GBK[3834] := 16#52B0;
   // UNICODE_TO_GBK[3835] := 16#84B9;
   // UNICODE_TO_GBK[3836] := 16#52B1;
   // UNICODE_TO_GBK[3837] := 16#C0F8;
   // UNICODE_TO_GBK[3838] := 16#52B2;
   // UNICODE_TO_GBK[3839] := 16#BEA2;
   // UNICODE_TO_GBK[3840] := 16#52B3;
   // UNICODE_TO_GBK[3841] := 16#C0CD;
   // UNICODE_TO_GBK[3842] := 16#52B4;
   // UNICODE_TO_GBK[3843] := 16#84BA;
   // UNICODE_TO_GBK[3844] := 16#52B5;
   // UNICODE_TO_GBK[3845] := 16#84BB;
   // UNICODE_TO_GBK[3846] := 16#52B6;
   // UNICODE_TO_GBK[3847] := 16#84BC;
   // UNICODE_TO_GBK[3848] := 16#52B7;
   // UNICODE_TO_GBK[3849] := 16#84BD;
   // UNICODE_TO_GBK[3850] := 16#52B8;
   // UNICODE_TO_GBK[3851] := 16#84BE;
   // UNICODE_TO_GBK[3852] := 16#52B9;
   // UNICODE_TO_GBK[3853] := 16#84BF;
   // UNICODE_TO_GBK[3854] := 16#52BA;
   // UNICODE_TO_GBK[3855] := 16#84C0;
   // UNICODE_TO_GBK[3856] := 16#52BB;
   // UNICODE_TO_GBK[3857] := 16#84C1;
   // UNICODE_TO_GBK[3858] := 16#52BC;
   // UNICODE_TO_GBK[3859] := 16#84C2;
   // UNICODE_TO_GBK[3860] := 16#52BD;
   // UNICODE_TO_GBK[3861] := 16#84C3;
   // UNICODE_TO_GBK[3862] := 16#52BE;
   // UNICODE_TO_GBK[3863] := 16#DBC0;
   // UNICODE_TO_GBK[3864] := 16#52BF;
   // UNICODE_TO_GBK[3865] := 16#CAC6;
   // UNICODE_TO_GBK[3866] := 16#52C0;
   // UNICODE_TO_GBK[3867] := 16#84C4;
   // UNICODE_TO_GBK[3868] := 16#52C1;
   // UNICODE_TO_GBK[3869] := 16#84C5;
   // UNICODE_TO_GBK[3870] := 16#52C2;
   // UNICODE_TO_GBK[3871] := 16#84C6;
   // UNICODE_TO_GBK[3872] := 16#52C3;
   // UNICODE_TO_GBK[3873] := 16#B2AA;
   // UNICODE_TO_GBK[3874] := 16#52C4;
   // UNICODE_TO_GBK[3875] := 16#84C7;
   // UNICODE_TO_GBK[3876] := 16#52C5;
   // UNICODE_TO_GBK[3877] := 16#84C8;
   // UNICODE_TO_GBK[3878] := 16#52C6;
   // UNICODE_TO_GBK[3879] := 16#84C9;
   // UNICODE_TO_GBK[3880] := 16#52C7;
   // UNICODE_TO_GBK[3881] := 16#D3C2;
   // UNICODE_TO_GBK[3882] := 16#52C8;
   // UNICODE_TO_GBK[3883] := 16#84CA;
   // UNICODE_TO_GBK[3884] := 16#52C9;
   // UNICODE_TO_GBK[3885] := 16#C3E3;
   // UNICODE_TO_GBK[3886] := 16#52CA;
   // UNICODE_TO_GBK[3887] := 16#84CB;
   // UNICODE_TO_GBK[3888] := 16#52CB;
   // UNICODE_TO_GBK[3889] := 16#D1AB;
   // UNICODE_TO_GBK[3890] := 16#52CC;
   // UNICODE_TO_GBK[3891] := 16#84CC;
   // UNICODE_TO_GBK[3892] := 16#52CD;
   // UNICODE_TO_GBK[3893] := 16#84CD;
   // UNICODE_TO_GBK[3894] := 16#52CE;
   // UNICODE_TO_GBK[3895] := 16#84CE;
   // UNICODE_TO_GBK[3896] := 16#52CF;
   // UNICODE_TO_GBK[3897] := 16#84CF;
   // UNICODE_TO_GBK[3898] := 16#52D0;
   // UNICODE_TO_GBK[3899] := 16#DBC2;
   // UNICODE_TO_GBK[3900] := 16#52D1;
   // UNICODE_TO_GBK[3901] := 16#84D0;
   // UNICODE_TO_GBK[3902] := 16#52D2;
   // UNICODE_TO_GBK[3903] := 16#C0D5;
   // UNICODE_TO_GBK[3904] := 16#52D3;
   // UNICODE_TO_GBK[3905] := 16#84D1;
   // UNICODE_TO_GBK[3906] := 16#52D4;
   // UNICODE_TO_GBK[3907] := 16#84D2;
   // UNICODE_TO_GBK[3908] := 16#52D5;
   // UNICODE_TO_GBK[3909] := 16#84D3;
   // UNICODE_TO_GBK[3910] := 16#52D6;
   // UNICODE_TO_GBK[3911] := 16#DBC3;
   // UNICODE_TO_GBK[3912] := 16#52D7;
   // UNICODE_TO_GBK[3913] := 16#84D4;
   // UNICODE_TO_GBK[3914] := 16#52D8;
   // UNICODE_TO_GBK[3915] := 16#BFB1;
   // UNICODE_TO_GBK[3916] := 16#52D9;
   // UNICODE_TO_GBK[3917] := 16#84D5;
   // UNICODE_TO_GBK[3918] := 16#52DA;
   // UNICODE_TO_GBK[3919] := 16#84D6;
   // UNICODE_TO_GBK[3920] := 16#52DB;
   // UNICODE_TO_GBK[3921] := 16#84D7;
   // UNICODE_TO_GBK[3922] := 16#52DC;
   // UNICODE_TO_GBK[3923] := 16#84D8;
   // UNICODE_TO_GBK[3924] := 16#52DD;
   // UNICODE_TO_GBK[3925] := 16#84D9;
   // UNICODE_TO_GBK[3926] := 16#52DE;
   // UNICODE_TO_GBK[3927] := 16#84DA;
   // UNICODE_TO_GBK[3928] := 16#52DF;
   // UNICODE_TO_GBK[3929] := 16#C4BC;
   // UNICODE_TO_GBK[3930] := 16#52E0;
   // UNICODE_TO_GBK[3931] := 16#84DB;
   // UNICODE_TO_GBK[3932] := 16#52E1;
   // UNICODE_TO_GBK[3933] := 16#84DC;
   // UNICODE_TO_GBK[3934] := 16#52E2;
   // UNICODE_TO_GBK[3935] := 16#84DD;
   // UNICODE_TO_GBK[3936] := 16#52E3;
   // UNICODE_TO_GBK[3937] := 16#84DE;
   // UNICODE_TO_GBK[3938] := 16#52E4;
   // UNICODE_TO_GBK[3939] := 16#C7DA;
   // UNICODE_TO_GBK[3940] := 16#52E5;
   // UNICODE_TO_GBK[3941] := 16#84DF;
   // UNICODE_TO_GBK[3942] := 16#52E6;
   // UNICODE_TO_GBK[3943] := 16#84E0;
   // UNICODE_TO_GBK[3944] := 16#52E7;
   // UNICODE_TO_GBK[3945] := 16#84E1;
   // UNICODE_TO_GBK[3946] := 16#52E8;
   // UNICODE_TO_GBK[3947] := 16#84E2;
   // UNICODE_TO_GBK[3948] := 16#52E9;
   // UNICODE_TO_GBK[3949] := 16#84E3;
   // UNICODE_TO_GBK[3950] := 16#52EA;
   // UNICODE_TO_GBK[3951] := 16#84E4;
   // UNICODE_TO_GBK[3952] := 16#52EB;
   // UNICODE_TO_GBK[3953] := 16#84E5;
   // UNICODE_TO_GBK[3954] := 16#52EC;
   // UNICODE_TO_GBK[3955] := 16#84E6;
   // UNICODE_TO_GBK[3956] := 16#52ED;
   // UNICODE_TO_GBK[3957] := 16#84E7;
   // UNICODE_TO_GBK[3958] := 16#52EE;
   // UNICODE_TO_GBK[3959] := 16#84E8;
   // UNICODE_TO_GBK[3960] := 16#52EF;
   // UNICODE_TO_GBK[3961] := 16#84E9;
   // UNICODE_TO_GBK[3962] := 16#52F0;
   // UNICODE_TO_GBK[3963] := 16#DBC4;
   // UNICODE_TO_GBK[3964] := 16#52F1;
   // UNICODE_TO_GBK[3965] := 16#84EA;
   // UNICODE_TO_GBK[3966] := 16#52F2;
   // UNICODE_TO_GBK[3967] := 16#84EB;
   // UNICODE_TO_GBK[3968] := 16#52F3;
   // UNICODE_TO_GBK[3969] := 16#84EC;
   // UNICODE_TO_GBK[3970] := 16#52F4;
   // UNICODE_TO_GBK[3971] := 16#84ED;
   // UNICODE_TO_GBK[3972] := 16#52F5;
   // UNICODE_TO_GBK[3973] := 16#84EE;
   // UNICODE_TO_GBK[3974] := 16#52F6;
   // UNICODE_TO_GBK[3975] := 16#84EF;
   // UNICODE_TO_GBK[3976] := 16#52F7;
   // UNICODE_TO_GBK[3977] := 16#84F0;
   // UNICODE_TO_GBK[3978] := 16#52F8;
   // UNICODE_TO_GBK[3979] := 16#84F1;
   // UNICODE_TO_GBK[3980] := 16#52F9;
   // UNICODE_TO_GBK[3981] := 16#D9E8;
   // UNICODE_TO_GBK[3982] := 16#52FA;
   // UNICODE_TO_GBK[3983] := 16#C9D7;
   // UNICODE_TO_GBK[3984] := 16#52FB;
   // UNICODE_TO_GBK[3985] := 16#84F2;
   // UNICODE_TO_GBK[3986] := 16#52FC;
   // UNICODE_TO_GBK[3987] := 16#84F3;
   // UNICODE_TO_GBK[3988] := 16#52FD;
   // UNICODE_TO_GBK[3989] := 16#84F4;
   // UNICODE_TO_GBK[3990] := 16#52FE;
   // UNICODE_TO_GBK[3991] := 16#B9B4;
   // UNICODE_TO_GBK[3992] := 16#52FF;
   // UNICODE_TO_GBK[3993] := 16#CEF0;
   // UNICODE_TO_GBK[3994] := 16#5300;
   // UNICODE_TO_GBK[3995] := 16#D4C8;
   // UNICODE_TO_GBK[3996] := 16#5301;
   // UNICODE_TO_GBK[3997] := 16#84F5;
   // UNICODE_TO_GBK[3998] := 16#5302;
   // UNICODE_TO_GBK[3999] := 16#84F6;
   // UNICODE_TO_GBK[4000] := 16#5303;
   // UNICODE_TO_GBK[4001] := 16#84F7;
   // UNICODE_TO_GBK[4002] := 16#5304;
   // UNICODE_TO_GBK[4003] := 16#84F8;
   // UNICODE_TO_GBK[4004] := 16#5305;
   // UNICODE_TO_GBK[4005] := 16#B0FC;
   // UNICODE_TO_GBK[4006] := 16#5306;
   // UNICODE_TO_GBK[4007] := 16#B4D2;
   // UNICODE_TO_GBK[4008] := 16#5307;
   // UNICODE_TO_GBK[4009] := 16#84F9;
   // UNICODE_TO_GBK[4010] := 16#5308;
   // UNICODE_TO_GBK[4011] := 16#D0D9;
   // UNICODE_TO_GBK[4012] := 16#5309;
   // UNICODE_TO_GBK[4013] := 16#84FA;
   // UNICODE_TO_GBK[4014] := 16#530A;
   // UNICODE_TO_GBK[4015] := 16#84FB;
   // UNICODE_TO_GBK[4016] := 16#530B;
   // UNICODE_TO_GBK[4017] := 16#84FC;
   // UNICODE_TO_GBK[4018] := 16#530C;
   // UNICODE_TO_GBK[4019] := 16#84FD;
   // UNICODE_TO_GBK[4020] := 16#530D;
   // UNICODE_TO_GBK[4021] := 16#D9E9;
   // UNICODE_TO_GBK[4022] := 16#530E;
   // UNICODE_TO_GBK[4023] := 16#84FE;
   // UNICODE_TO_GBK[4024] := 16#530F;
   // UNICODE_TO_GBK[4025] := 16#DECB;
   // UNICODE_TO_GBK[4026] := 16#5310;
   // UNICODE_TO_GBK[4027] := 16#D9EB;
   // UNICODE_TO_GBK[4028] := 16#5311;
   // UNICODE_TO_GBK[4029] := 16#8540;
   // UNICODE_TO_GBK[4030] := 16#5312;
   // UNICODE_TO_GBK[4031] := 16#8541;
   // UNICODE_TO_GBK[4032] := 16#5313;
   // UNICODE_TO_GBK[4033] := 16#8542;
   // UNICODE_TO_GBK[4034] := 16#5314;
   // UNICODE_TO_GBK[4035] := 16#8543;
   // UNICODE_TO_GBK[4036] := 16#5315;
   // UNICODE_TO_GBK[4037] := 16#D8B0;
   // UNICODE_TO_GBK[4038] := 16#5316;
   // UNICODE_TO_GBK[4039] := 16#BBAF;
   // UNICODE_TO_GBK[4040] := 16#5317;
   // UNICODE_TO_GBK[4041] := 16#B1B1;
   // UNICODE_TO_GBK[4042] := 16#5318;
   // UNICODE_TO_GBK[4043] := 16#8544;
   // UNICODE_TO_GBK[4044] := 16#5319;
   // UNICODE_TO_GBK[4045] := 16#B3D7;
   // UNICODE_TO_GBK[4046] := 16#531A;
   // UNICODE_TO_GBK[4047] := 16#D8CE;
   // UNICODE_TO_GBK[4048] := 16#531B;
   // UNICODE_TO_GBK[4049] := 16#8545;
   // UNICODE_TO_GBK[4050] := 16#531C;
   // UNICODE_TO_GBK[4051] := 16#8546;
   // UNICODE_TO_GBK[4052] := 16#531D;
   // UNICODE_TO_GBK[4053] := 16#D4D1;
   // UNICODE_TO_GBK[4054] := 16#531E;
   // UNICODE_TO_GBK[4055] := 16#8547;
   // UNICODE_TO_GBK[4056] := 16#531F;
   // UNICODE_TO_GBK[4057] := 16#8548;
   // UNICODE_TO_GBK[4058] := 16#5320;
   // UNICODE_TO_GBK[4059] := 16#BDB3;
   // UNICODE_TO_GBK[4060] := 16#5321;
   // UNICODE_TO_GBK[4061] := 16#BFEF;
   // UNICODE_TO_GBK[4062] := 16#5322;
   // UNICODE_TO_GBK[4063] := 16#8549;
   // UNICODE_TO_GBK[4064] := 16#5323;
   // UNICODE_TO_GBK[4065] := 16#CFBB;
   // UNICODE_TO_GBK[4066] := 16#5324;
   // UNICODE_TO_GBK[4067] := 16#854A;
   // UNICODE_TO_GBK[4068] := 16#5325;
   // UNICODE_TO_GBK[4069] := 16#854B;
   // UNICODE_TO_GBK[4070] := 16#5326;
   // UNICODE_TO_GBK[4071] := 16#D8D0;
   // UNICODE_TO_GBK[4072] := 16#5327;
   // UNICODE_TO_GBK[4073] := 16#854C;
   // UNICODE_TO_GBK[4074] := 16#5328;
   // UNICODE_TO_GBK[4075] := 16#854D;
   // UNICODE_TO_GBK[4076] := 16#5329;
   // UNICODE_TO_GBK[4077] := 16#854E;
   // UNICODE_TO_GBK[4078] := 16#532A;
   // UNICODE_TO_GBK[4079] := 16#B7CB;
   // UNICODE_TO_GBK[4080] := 16#532B;
   // UNICODE_TO_GBK[4081] := 16#854F;
   // UNICODE_TO_GBK[4082] := 16#532C;
   // UNICODE_TO_GBK[4083] := 16#8550;
   // UNICODE_TO_GBK[4084] := 16#532D;
   // UNICODE_TO_GBK[4085] := 16#8551;
   // UNICODE_TO_GBK[4086] := 16#532E;
   // UNICODE_TO_GBK[4087] := 16#D8D1;
   // UNICODE_TO_GBK[4088] := 16#532F;
   // UNICODE_TO_GBK[4089] := 16#8552;
   // UNICODE_TO_GBK[4090] := 16#5330;
   // UNICODE_TO_GBK[4091] := 16#8553;
   // UNICODE_TO_GBK[4092] := 16#5331;
   // UNICODE_TO_GBK[4093] := 16#8554;
   // UNICODE_TO_GBK[4094] := 16#5332;
   // UNICODE_TO_GBK[4095] := 16#8555;
   // UNICODE_TO_GBK[4096] := 16#5333;
   // UNICODE_TO_GBK[4097] := 16#8556;
   // UNICODE_TO_GBK[4098] := 16#5334;
   // UNICODE_TO_GBK[4099] := 16#8557;
   // UNICODE_TO_GBK[4100] := 16#5335;
   // UNICODE_TO_GBK[4101] := 16#8558;
   // UNICODE_TO_GBK[4102] := 16#5336;
   // UNICODE_TO_GBK[4103] := 16#8559;
   // UNICODE_TO_GBK[4104] := 16#5337;
   // UNICODE_TO_GBK[4105] := 16#855A;
   // UNICODE_TO_GBK[4106] := 16#5338;
   // UNICODE_TO_GBK[4107] := 16#855B;
   // UNICODE_TO_GBK[4108] := 16#5339;
   // UNICODE_TO_GBK[4109] := 16#C6A5;
   // UNICODE_TO_GBK[4110] := 16#533A;
   // UNICODE_TO_GBK[4111] := 16#C7F8;
   // UNICODE_TO_GBK[4112] := 16#533B;
   // UNICODE_TO_GBK[4113] := 16#D2BD;
   // UNICODE_TO_GBK[4114] := 16#533C;
   // UNICODE_TO_GBK[4115] := 16#855C;
   // UNICODE_TO_GBK[4116] := 16#533D;
   // UNICODE_TO_GBK[4117] := 16#855D;
   // UNICODE_TO_GBK[4118] := 16#533E;
   // UNICODE_TO_GBK[4119] := 16#D8D2;
   // UNICODE_TO_GBK[4120] := 16#533F;
   // UNICODE_TO_GBK[4121] := 16#C4E4;
   // UNICODE_TO_GBK[4122] := 16#5340;
   // UNICODE_TO_GBK[4123] := 16#855E;
   // UNICODE_TO_GBK[4124] := 16#5341;
   // UNICODE_TO_GBK[4125] := 16#CAAE;
   // UNICODE_TO_GBK[4126] := 16#5342;
   // UNICODE_TO_GBK[4127] := 16#855F;
   // UNICODE_TO_GBK[4128] := 16#5343;
   // UNICODE_TO_GBK[4129] := 16#C7A7;
   // UNICODE_TO_GBK[4130] := 16#5344;
   // UNICODE_TO_GBK[4131] := 16#8560;
   // UNICODE_TO_GBK[4132] := 16#5345;
   // UNICODE_TO_GBK[4133] := 16#D8A6;
   // UNICODE_TO_GBK[4134] := 16#5346;
   // UNICODE_TO_GBK[4135] := 16#8561;
   // UNICODE_TO_GBK[4136] := 16#5347;
   // UNICODE_TO_GBK[4137] := 16#C9FD;
   // UNICODE_TO_GBK[4138] := 16#5348;
   // UNICODE_TO_GBK[4139] := 16#CEE7;
   // UNICODE_TO_GBK[4140] := 16#5349;
   // UNICODE_TO_GBK[4141] := 16#BBDC;
   // UNICODE_TO_GBK[4142] := 16#534A;
   // UNICODE_TO_GBK[4143] := 16#B0EB;
   // UNICODE_TO_GBK[4144] := 16#534B;
   // UNICODE_TO_GBK[4145] := 16#8562;
   // UNICODE_TO_GBK[4146] := 16#534C;
   // UNICODE_TO_GBK[4147] := 16#8563;
   // UNICODE_TO_GBK[4148] := 16#534D;
   // UNICODE_TO_GBK[4149] := 16#8564;
   // UNICODE_TO_GBK[4150] := 16#534E;
   // UNICODE_TO_GBK[4151] := 16#BBAA;
   // UNICODE_TO_GBK[4152] := 16#534F;
   // UNICODE_TO_GBK[4153] := 16#D0AD;
   // UNICODE_TO_GBK[4154] := 16#5350;
   // UNICODE_TO_GBK[4155] := 16#8565;
   // UNICODE_TO_GBK[4156] := 16#5351;
   // UNICODE_TO_GBK[4157] := 16#B1B0;
   // UNICODE_TO_GBK[4158] := 16#5352;
   // UNICODE_TO_GBK[4159] := 16#D7E4;
   // UNICODE_TO_GBK[4160] := 16#5353;
   // UNICODE_TO_GBK[4161] := 16#D7BF;
   // UNICODE_TO_GBK[4162] := 16#5354;
   // UNICODE_TO_GBK[4163] := 16#8566;
   // UNICODE_TO_GBK[4164] := 16#5355;
   // UNICODE_TO_GBK[4165] := 16#B5A5;
   // UNICODE_TO_GBK[4166] := 16#5356;
   // UNICODE_TO_GBK[4167] := 16#C2F4;
   // UNICODE_TO_GBK[4168] := 16#5357;
   // UNICODE_TO_GBK[4169] := 16#C4CF;
   // UNICODE_TO_GBK[4170] := 16#5358;
   // UNICODE_TO_GBK[4171] := 16#8567;
   // UNICODE_TO_GBK[4172] := 16#5359;
   // UNICODE_TO_GBK[4173] := 16#8568;
   // UNICODE_TO_GBK[4174] := 16#535A;
   // UNICODE_TO_GBK[4175] := 16#B2A9;
   // UNICODE_TO_GBK[4176] := 16#535B;
   // UNICODE_TO_GBK[4177] := 16#8569;
   // UNICODE_TO_GBK[4178] := 16#535C;
   // UNICODE_TO_GBK[4179] := 16#B2B7;
   // UNICODE_TO_GBK[4180] := 16#535D;
   // UNICODE_TO_GBK[4181] := 16#856A;
   // UNICODE_TO_GBK[4182] := 16#535E;
   // UNICODE_TO_GBK[4183] := 16#B1E5;
   // UNICODE_TO_GBK[4184] := 16#535F;
   // UNICODE_TO_GBK[4185] := 16#DFB2;
   // UNICODE_TO_GBK[4186] := 16#5360;
   // UNICODE_TO_GBK[4187] := 16#D5BC;
   // UNICODE_TO_GBK[4188] := 16#5361;
   // UNICODE_TO_GBK[4189] := 16#BFA8;
   // UNICODE_TO_GBK[4190] := 16#5362;
   // UNICODE_TO_GBK[4191] := 16#C2AC;
   // UNICODE_TO_GBK[4192] := 16#5363;
   // UNICODE_TO_GBK[4193] := 16#D8D5;
   // UNICODE_TO_GBK[4194] := 16#5364;
   // UNICODE_TO_GBK[4195] := 16#C2B1;
   // UNICODE_TO_GBK[4196] := 16#5365;
   // UNICODE_TO_GBK[4197] := 16#856B;
   // UNICODE_TO_GBK[4198] := 16#5366;
   // UNICODE_TO_GBK[4199] := 16#D8D4;
   // UNICODE_TO_GBK[4200] := 16#5367;
   // UNICODE_TO_GBK[4201] := 16#CED4;
   // UNICODE_TO_GBK[4202] := 16#5368;
   // UNICODE_TO_GBK[4203] := 16#856C;
   // UNICODE_TO_GBK[4204] := 16#5369;
   // UNICODE_TO_GBK[4205] := 16#DAE0;
   // UNICODE_TO_GBK[4206] := 16#536A;
   // UNICODE_TO_GBK[4207] := 16#856D;
   // UNICODE_TO_GBK[4208] := 16#536B;
   // UNICODE_TO_GBK[4209] := 16#CEC0;
   // UNICODE_TO_GBK[4210] := 16#536C;
   // UNICODE_TO_GBK[4211] := 16#856E;
   // UNICODE_TO_GBK[4212] := 16#536D;
   // UNICODE_TO_GBK[4213] := 16#856F;
   // UNICODE_TO_GBK[4214] := 16#536E;
   // UNICODE_TO_GBK[4215] := 16#D8B4;
   // UNICODE_TO_GBK[4216] := 16#536F;
   // UNICODE_TO_GBK[4217] := 16#C3AE;
   // UNICODE_TO_GBK[4218] := 16#5370;
   // UNICODE_TO_GBK[4219] := 16#D3A1;
   // UNICODE_TO_GBK[4220] := 16#5371;
   // UNICODE_TO_GBK[4221] := 16#CEA3;
   // UNICODE_TO_GBK[4222] := 16#5372;
   // UNICODE_TO_GBK[4223] := 16#8570;
   // UNICODE_TO_GBK[4224] := 16#5373;
   // UNICODE_TO_GBK[4225] := 16#BCB4;
   // UNICODE_TO_GBK[4226] := 16#5374;
   // UNICODE_TO_GBK[4227] := 16#C8B4;
   // UNICODE_TO_GBK[4228] := 16#5375;
   // UNICODE_TO_GBK[4229] := 16#C2D1;
   // UNICODE_TO_GBK[4230] := 16#5376;
   // UNICODE_TO_GBK[4231] := 16#8571;
   // UNICODE_TO_GBK[4232] := 16#5377;
   // UNICODE_TO_GBK[4233] := 16#BEED;
   // UNICODE_TO_GBK[4234] := 16#5378;
   // UNICODE_TO_GBK[4235] := 16#D0B6;
   // UNICODE_TO_GBK[4236] := 16#5379;
   // UNICODE_TO_GBK[4237] := 16#8572;
   // UNICODE_TO_GBK[4238] := 16#537A;
   // UNICODE_TO_GBK[4239] := 16#DAE1;
   // UNICODE_TO_GBK[4240] := 16#537B;
   // UNICODE_TO_GBK[4241] := 16#8573;
   // UNICODE_TO_GBK[4242] := 16#537C;
   // UNICODE_TO_GBK[4243] := 16#8574;
   // UNICODE_TO_GBK[4244] := 16#537D;
   // UNICODE_TO_GBK[4245] := 16#8575;
   // UNICODE_TO_GBK[4246] := 16#537E;
   // UNICODE_TO_GBK[4247] := 16#8576;
   // UNICODE_TO_GBK[4248] := 16#537F;
   // UNICODE_TO_GBK[4249] := 16#C7E4;
   // UNICODE_TO_GBK[4250] := 16#5380;
   // UNICODE_TO_GBK[4251] := 16#8577;
   // UNICODE_TO_GBK[4252] := 16#5381;
   // UNICODE_TO_GBK[4253] := 16#8578;
   // UNICODE_TO_GBK[4254] := 16#5382;
   // UNICODE_TO_GBK[4255] := 16#B3A7;
   // UNICODE_TO_GBK[4256] := 16#5383;
   // UNICODE_TO_GBK[4257] := 16#8579;
   // UNICODE_TO_GBK[4258] := 16#5384;
   // UNICODE_TO_GBK[4259] := 16#B6F2;
   // UNICODE_TO_GBK[4260] := 16#5385;
   // UNICODE_TO_GBK[4261] := 16#CCFC;
   // UNICODE_TO_GBK[4262] := 16#5386;
   // UNICODE_TO_GBK[4263] := 16#C0FA;
   // UNICODE_TO_GBK[4264] := 16#5387;
   // UNICODE_TO_GBK[4265] := 16#857A;
   // UNICODE_TO_GBK[4266] := 16#5388;
   // UNICODE_TO_GBK[4267] := 16#857B;
   // UNICODE_TO_GBK[4268] := 16#5389;
   // UNICODE_TO_GBK[4269] := 16#C0F7;
   // UNICODE_TO_GBK[4270] := 16#538A;
   // UNICODE_TO_GBK[4271] := 16#857C;
   // UNICODE_TO_GBK[4272] := 16#538B;
   // UNICODE_TO_GBK[4273] := 16#D1B9;
   // UNICODE_TO_GBK[4274] := 16#538C;
   // UNICODE_TO_GBK[4275] := 16#D1E1;
   // UNICODE_TO_GBK[4276] := 16#538D;
   // UNICODE_TO_GBK[4277] := 16#D8C7;
   // UNICODE_TO_GBK[4278] := 16#538E;
   // UNICODE_TO_GBK[4279] := 16#857D;
   // UNICODE_TO_GBK[4280] := 16#538F;
   // UNICODE_TO_GBK[4281] := 16#857E;
   // UNICODE_TO_GBK[4282] := 16#5390;
   // UNICODE_TO_GBK[4283] := 16#8580;
   // UNICODE_TO_GBK[4284] := 16#5391;
   // UNICODE_TO_GBK[4285] := 16#8581;
   // UNICODE_TO_GBK[4286] := 16#5392;
   // UNICODE_TO_GBK[4287] := 16#8582;
   // UNICODE_TO_GBK[4288] := 16#5393;
   // UNICODE_TO_GBK[4289] := 16#8583;
   // UNICODE_TO_GBK[4290] := 16#5394;
   // UNICODE_TO_GBK[4291] := 16#8584;
   // UNICODE_TO_GBK[4292] := 16#5395;
   // UNICODE_TO_GBK[4293] := 16#B2DE;
   // UNICODE_TO_GBK[4294] := 16#5396;
   // UNICODE_TO_GBK[4295] := 16#8585;
   // UNICODE_TO_GBK[4296] := 16#5397;
   // UNICODE_TO_GBK[4297] := 16#8586;
   // UNICODE_TO_GBK[4298] := 16#5398;
   // UNICODE_TO_GBK[4299] := 16#C0E5;
   // UNICODE_TO_GBK[4300] := 16#5399;
   // UNICODE_TO_GBK[4301] := 16#8587;
   // UNICODE_TO_GBK[4302] := 16#539A;
   // UNICODE_TO_GBK[4303] := 16#BAF1;
   // UNICODE_TO_GBK[4304] := 16#539B;
   // UNICODE_TO_GBK[4305] := 16#8588;
   // UNICODE_TO_GBK[4306] := 16#539C;
   // UNICODE_TO_GBK[4307] := 16#8589;
   // UNICODE_TO_GBK[4308] := 16#539D;
   // UNICODE_TO_GBK[4309] := 16#D8C8;
   // UNICODE_TO_GBK[4310] := 16#539E;
   // UNICODE_TO_GBK[4311] := 16#858A;
   // UNICODE_TO_GBK[4312] := 16#539F;
   // UNICODE_TO_GBK[4313] := 16#D4AD;
   // UNICODE_TO_GBK[4314] := 16#53A0;
   // UNICODE_TO_GBK[4315] := 16#858B;
   // UNICODE_TO_GBK[4316] := 16#53A1;
   // UNICODE_TO_GBK[4317] := 16#858C;
   // UNICODE_TO_GBK[4318] := 16#53A2;
   // UNICODE_TO_GBK[4319] := 16#CFE1;
   // UNICODE_TO_GBK[4320] := 16#53A3;
   // UNICODE_TO_GBK[4321] := 16#D8C9;
   // UNICODE_TO_GBK[4322] := 16#53A4;
   // UNICODE_TO_GBK[4323] := 16#858D;
   // UNICODE_TO_GBK[4324] := 16#53A5;
   // UNICODE_TO_GBK[4325] := 16#D8CA;
   // UNICODE_TO_GBK[4326] := 16#53A6;
   // UNICODE_TO_GBK[4327] := 16#CFC3;
   // UNICODE_TO_GBK[4328] := 16#53A7;
   // UNICODE_TO_GBK[4329] := 16#858E;
   // UNICODE_TO_GBK[4330] := 16#53A8;
   // UNICODE_TO_GBK[4331] := 16#B3F8;
   // UNICODE_TO_GBK[4332] := 16#53A9;
   // UNICODE_TO_GBK[4333] := 16#BEC7;
   // UNICODE_TO_GBK[4334] := 16#53AA;
   // UNICODE_TO_GBK[4335] := 16#858F;
   // UNICODE_TO_GBK[4336] := 16#53AB;
   // UNICODE_TO_GBK[4337] := 16#8590;
   // UNICODE_TO_GBK[4338] := 16#53AC;
   // UNICODE_TO_GBK[4339] := 16#8591;
   // UNICODE_TO_GBK[4340] := 16#53AD;
   // UNICODE_TO_GBK[4341] := 16#8592;
   // UNICODE_TO_GBK[4342] := 16#53AE;
   // UNICODE_TO_GBK[4343] := 16#D8CB;
   // UNICODE_TO_GBK[4344] := 16#53AF;
   // UNICODE_TO_GBK[4345] := 16#8593;
   // UNICODE_TO_GBK[4346] := 16#53B0;
   // UNICODE_TO_GBK[4347] := 16#8594;
   // UNICODE_TO_GBK[4348] := 16#53B1;
   // UNICODE_TO_GBK[4349] := 16#8595;
   // UNICODE_TO_GBK[4350] := 16#53B2;
   // UNICODE_TO_GBK[4351] := 16#8596;
   // UNICODE_TO_GBK[4352] := 16#53B3;
   // UNICODE_TO_GBK[4353] := 16#8597;
   // UNICODE_TO_GBK[4354] := 16#53B4;
   // UNICODE_TO_GBK[4355] := 16#8598;
   // UNICODE_TO_GBK[4356] := 16#53B5;
   // UNICODE_TO_GBK[4357] := 16#8599;
   // UNICODE_TO_GBK[4358] := 16#53B6;
   // UNICODE_TO_GBK[4359] := 16#DBCC;
   // UNICODE_TO_GBK[4360] := 16#53B7;
   // UNICODE_TO_GBK[4361] := 16#859A;
   // UNICODE_TO_GBK[4362] := 16#53B8;
   // UNICODE_TO_GBK[4363] := 16#859B;
   // UNICODE_TO_GBK[4364] := 16#53B9;
   // UNICODE_TO_GBK[4365] := 16#859C;
   // UNICODE_TO_GBK[4366] := 16#53BA;
   // UNICODE_TO_GBK[4367] := 16#859D;
   // UNICODE_TO_GBK[4368] := 16#53BB;
   // UNICODE_TO_GBK[4369] := 16#C8A5;
   // UNICODE_TO_GBK[4370] := 16#53BC;
   // UNICODE_TO_GBK[4371] := 16#859E;
   // UNICODE_TO_GBK[4372] := 16#53BD;
   // UNICODE_TO_GBK[4373] := 16#859F;
   // UNICODE_TO_GBK[4374] := 16#53BE;
   // UNICODE_TO_GBK[4375] := 16#85A0;
   // UNICODE_TO_GBK[4376] := 16#53BF;
   // UNICODE_TO_GBK[4377] := 16#CFD8;
   // UNICODE_TO_GBK[4378] := 16#53C0;
   // UNICODE_TO_GBK[4379] := 16#85A1;
   // UNICODE_TO_GBK[4380] := 16#53C1;
   // UNICODE_TO_GBK[4381] := 16#C8FE;
   // UNICODE_TO_GBK[4382] := 16#53C2;
   // UNICODE_TO_GBK[4383] := 16#B2CE;
   // UNICODE_TO_GBK[4384] := 16#53C3;
   // UNICODE_TO_GBK[4385] := 16#85A2;
   // UNICODE_TO_GBK[4386] := 16#53C4;
   // UNICODE_TO_GBK[4387] := 16#85A3;
   // UNICODE_TO_GBK[4388] := 16#53C5;
   // UNICODE_TO_GBK[4389] := 16#85A4;
   // UNICODE_TO_GBK[4390] := 16#53C6;
   // UNICODE_TO_GBK[4391] := 16#85A5;
   // UNICODE_TO_GBK[4392] := 16#53C7;
   // UNICODE_TO_GBK[4393] := 16#85A6;
   // UNICODE_TO_GBK[4394] := 16#53C8;
   // UNICODE_TO_GBK[4395] := 16#D3D6;
   // UNICODE_TO_GBK[4396] := 16#53C9;
   // UNICODE_TO_GBK[4397] := 16#B2E6;
   // UNICODE_TO_GBK[4398] := 16#53CA;
   // UNICODE_TO_GBK[4399] := 16#BCB0;
   // UNICODE_TO_GBK[4400] := 16#53CB;
   // UNICODE_TO_GBK[4401] := 16#D3D1;
   // UNICODE_TO_GBK[4402] := 16#53CC;
   // UNICODE_TO_GBK[4403] := 16#CBAB;
   // UNICODE_TO_GBK[4404] := 16#53CD;
   // UNICODE_TO_GBK[4405] := 16#B7B4;
   // UNICODE_TO_GBK[4406] := 16#53CE;
   // UNICODE_TO_GBK[4407] := 16#85A7;
   // UNICODE_TO_GBK[4408] := 16#53CF;
   // UNICODE_TO_GBK[4409] := 16#85A8;
   // UNICODE_TO_GBK[4410] := 16#53D0;
   // UNICODE_TO_GBK[4411] := 16#85A9;
   // UNICODE_TO_GBK[4412] := 16#53D1;
   // UNICODE_TO_GBK[4413] := 16#B7A2;
   // UNICODE_TO_GBK[4414] := 16#53D2;
   // UNICODE_TO_GBK[4415] := 16#85AA;
   // UNICODE_TO_GBK[4416] := 16#53D3;
   // UNICODE_TO_GBK[4417] := 16#85AB;
   // UNICODE_TO_GBK[4418] := 16#53D4;
   // UNICODE_TO_GBK[4419] := 16#CAE5;
   // UNICODE_TO_GBK[4420] := 16#53D5;
   // UNICODE_TO_GBK[4421] := 16#85AC;
   // UNICODE_TO_GBK[4422] := 16#53D6;
   // UNICODE_TO_GBK[4423] := 16#C8A1;
   // UNICODE_TO_GBK[4424] := 16#53D7;
   // UNICODE_TO_GBK[4425] := 16#CADC;
   // UNICODE_TO_GBK[4426] := 16#53D8;
   // UNICODE_TO_GBK[4427] := 16#B1E4;
   // UNICODE_TO_GBK[4428] := 16#53D9;
   // UNICODE_TO_GBK[4429] := 16#D0F0;
   // UNICODE_TO_GBK[4430] := 16#53DA;
   // UNICODE_TO_GBK[4431] := 16#85AD;
   // UNICODE_TO_GBK[4432] := 16#53DB;
   // UNICODE_TO_GBK[4433] := 16#C5D1;
   // UNICODE_TO_GBK[4434] := 16#53DC;
   // UNICODE_TO_GBK[4435] := 16#85AE;
   // UNICODE_TO_GBK[4436] := 16#53DD;
   // UNICODE_TO_GBK[4437] := 16#85AF;
   // UNICODE_TO_GBK[4438] := 16#53DE;
   // UNICODE_TO_GBK[4439] := 16#85B0;
   // UNICODE_TO_GBK[4440] := 16#53DF;
   // UNICODE_TO_GBK[4441] := 16#DBC5;
   // UNICODE_TO_GBK[4442] := 16#53E0;
   // UNICODE_TO_GBK[4443] := 16#B5FE;
   // UNICODE_TO_GBK[4444] := 16#53E1;
   // UNICODE_TO_GBK[4445] := 16#85B1;
   // UNICODE_TO_GBK[4446] := 16#53E2;
   // UNICODE_TO_GBK[4447] := 16#85B2;
   // UNICODE_TO_GBK[4448] := 16#53E3;
   // UNICODE_TO_GBK[4449] := 16#BFDA;
   // UNICODE_TO_GBK[4450] := 16#53E4;
   // UNICODE_TO_GBK[4451] := 16#B9C5;
   // UNICODE_TO_GBK[4452] := 16#53E5;
   // UNICODE_TO_GBK[4453] := 16#BEE4;
   // UNICODE_TO_GBK[4454] := 16#53E6;
   // UNICODE_TO_GBK[4455] := 16#C1ED;
   // UNICODE_TO_GBK[4456] := 16#53E7;
   // UNICODE_TO_GBK[4457] := 16#85B3;
   // UNICODE_TO_GBK[4458] := 16#53E8;
   // UNICODE_TO_GBK[4459] := 16#DFB6;
   // UNICODE_TO_GBK[4460] := 16#53E9;
   // UNICODE_TO_GBK[4461] := 16#DFB5;
   // UNICODE_TO_GBK[4462] := 16#53EA;
   // UNICODE_TO_GBK[4463] := 16#D6BB;
   // UNICODE_TO_GBK[4464] := 16#53EB;
   // UNICODE_TO_GBK[4465] := 16#BDD0;
   // UNICODE_TO_GBK[4466] := 16#53EC;
   // UNICODE_TO_GBK[4467] := 16#D5D9;
   // UNICODE_TO_GBK[4468] := 16#53ED;
   // UNICODE_TO_GBK[4469] := 16#B0C8;
   // UNICODE_TO_GBK[4470] := 16#53EE;
   // UNICODE_TO_GBK[4471] := 16#B6A3;
   // UNICODE_TO_GBK[4472] := 16#53EF;
   // UNICODE_TO_GBK[4473] := 16#BFC9;
   // UNICODE_TO_GBK[4474] := 16#53F0;
   // UNICODE_TO_GBK[4475] := 16#CCA8;
   // UNICODE_TO_GBK[4476] := 16#53F1;
   // UNICODE_TO_GBK[4477] := 16#DFB3;
   // UNICODE_TO_GBK[4478] := 16#53F2;
   // UNICODE_TO_GBK[4479] := 16#CAB7;
   // UNICODE_TO_GBK[4480] := 16#53F3;
   // UNICODE_TO_GBK[4481] := 16#D3D2;
   // UNICODE_TO_GBK[4482] := 16#53F4;
   // UNICODE_TO_GBK[4483] := 16#85B4;
   // UNICODE_TO_GBK[4484] := 16#53F5;
   // UNICODE_TO_GBK[4485] := 16#D8CF;
   // UNICODE_TO_GBK[4486] := 16#53F6;
   // UNICODE_TO_GBK[4487] := 16#D2B6;
   // UNICODE_TO_GBK[4488] := 16#53F7;
   // UNICODE_TO_GBK[4489] := 16#BAC5;
   // UNICODE_TO_GBK[4490] := 16#53F8;
   // UNICODE_TO_GBK[4491] := 16#CBBE;
   // UNICODE_TO_GBK[4492] := 16#53F9;
   // UNICODE_TO_GBK[4493] := 16#CCBE;
   // UNICODE_TO_GBK[4494] := 16#53FA;
   // UNICODE_TO_GBK[4495] := 16#85B5;
   // UNICODE_TO_GBK[4496] := 16#53FB;
   // UNICODE_TO_GBK[4497] := 16#DFB7;
   // UNICODE_TO_GBK[4498] := 16#53FC;
   // UNICODE_TO_GBK[4499] := 16#B5F0;
   // UNICODE_TO_GBK[4500] := 16#53FD;
   // UNICODE_TO_GBK[4501] := 16#DFB4;
   // UNICODE_TO_GBK[4502] := 16#53FE;
   // UNICODE_TO_GBK[4503] := 16#85B6;
   // UNICODE_TO_GBK[4504] := 16#53FF;
   // UNICODE_TO_GBK[4505] := 16#85B7;
   // UNICODE_TO_GBK[4506] := 16#5400;
   // UNICODE_TO_GBK[4507] := 16#85B8;
   // UNICODE_TO_GBK[4508] := 16#5401;
   // UNICODE_TO_GBK[4509] := 16#D3F5;
   // UNICODE_TO_GBK[4510] := 16#5402;
   // UNICODE_TO_GBK[4511] := 16#85B9;
   // UNICODE_TO_GBK[4512] := 16#5403;
   // UNICODE_TO_GBK[4513] := 16#B3D4;
   // UNICODE_TO_GBK[4514] := 16#5404;
   // UNICODE_TO_GBK[4515] := 16#B8F7;
   // UNICODE_TO_GBK[4516] := 16#5405;
   // UNICODE_TO_GBK[4517] := 16#85BA;
   // UNICODE_TO_GBK[4518] := 16#5406;
   // UNICODE_TO_GBK[4519] := 16#DFBA;
   // UNICODE_TO_GBK[4520] := 16#5407;
   // UNICODE_TO_GBK[4521] := 16#85BB;
   // UNICODE_TO_GBK[4522] := 16#5408;
   // UNICODE_TO_GBK[4523] := 16#BACF;
   // UNICODE_TO_GBK[4524] := 16#5409;
   // UNICODE_TO_GBK[4525] := 16#BCAA;
   // UNICODE_TO_GBK[4526] := 16#540A;
   // UNICODE_TO_GBK[4527] := 16#B5F5;
   // UNICODE_TO_GBK[4528] := 16#540B;
   // UNICODE_TO_GBK[4529] := 16#85BC;
   // UNICODE_TO_GBK[4530] := 16#540C;
   // UNICODE_TO_GBK[4531] := 16#CDAC;
   // UNICODE_TO_GBK[4532] := 16#540D;
   // UNICODE_TO_GBK[4533] := 16#C3FB;
   // UNICODE_TO_GBK[4534] := 16#540E;
   // UNICODE_TO_GBK[4535] := 16#BAF3;
   // UNICODE_TO_GBK[4536] := 16#540F;
   // UNICODE_TO_GBK[4537] := 16#C0F4;
   // UNICODE_TO_GBK[4538] := 16#5410;
   // UNICODE_TO_GBK[4539] := 16#CDC2;
   // UNICODE_TO_GBK[4540] := 16#5411;
   // UNICODE_TO_GBK[4541] := 16#CFF2;
   // UNICODE_TO_GBK[4542] := 16#5412;
   // UNICODE_TO_GBK[4543] := 16#DFB8;
   // UNICODE_TO_GBK[4544] := 16#5413;
   // UNICODE_TO_GBK[4545] := 16#CFC5;
   // UNICODE_TO_GBK[4546] := 16#5414;
   // UNICODE_TO_GBK[4547] := 16#85BD;
   // UNICODE_TO_GBK[4548] := 16#5415;
   // UNICODE_TO_GBK[4549] := 16#C2C0;
   // UNICODE_TO_GBK[4550] := 16#5416;
   // UNICODE_TO_GBK[4551] := 16#DFB9;
   // UNICODE_TO_GBK[4552] := 16#5417;
   // UNICODE_TO_GBK[4553] := 16#C2F0;
   // UNICODE_TO_GBK[4554] := 16#5418;
   // UNICODE_TO_GBK[4555] := 16#85BE;
   // UNICODE_TO_GBK[4556] := 16#5419;
   // UNICODE_TO_GBK[4557] := 16#85BF;
   // UNICODE_TO_GBK[4558] := 16#541A;
   // UNICODE_TO_GBK[4559] := 16#85C0;
   // UNICODE_TO_GBK[4560] := 16#541B;
   // UNICODE_TO_GBK[4561] := 16#BEFD;
   // UNICODE_TO_GBK[4562] := 16#541C;
   // UNICODE_TO_GBK[4563] := 16#85C1;
   // UNICODE_TO_GBK[4564] := 16#541D;
   // UNICODE_TO_GBK[4565] := 16#C1DF;
   // UNICODE_TO_GBK[4566] := 16#541E;
   // UNICODE_TO_GBK[4567] := 16#CDCC;
   // UNICODE_TO_GBK[4568] := 16#541F;
   // UNICODE_TO_GBK[4569] := 16#D2F7;
   // UNICODE_TO_GBK[4570] := 16#5420;
   // UNICODE_TO_GBK[4571] := 16#B7CD;
   // UNICODE_TO_GBK[4572] := 16#5421;
   // UNICODE_TO_GBK[4573] := 16#DFC1;
   // UNICODE_TO_GBK[4574] := 16#5422;
   // UNICODE_TO_GBK[4575] := 16#85C2;
   // UNICODE_TO_GBK[4576] := 16#5423;
   // UNICODE_TO_GBK[4577] := 16#DFC4;
   // UNICODE_TO_GBK[4578] := 16#5424;
   // UNICODE_TO_GBK[4579] := 16#85C3;
   // UNICODE_TO_GBK[4580] := 16#5425;
   // UNICODE_TO_GBK[4581] := 16#85C4;
   // UNICODE_TO_GBK[4582] := 16#5426;
   // UNICODE_TO_GBK[4583] := 16#B7F1;
   // UNICODE_TO_GBK[4584] := 16#5427;
   // UNICODE_TO_GBK[4585] := 16#B0C9;
   // UNICODE_TO_GBK[4586] := 16#5428;
   // UNICODE_TO_GBK[4587] := 16#B6D6;
   // UNICODE_TO_GBK[4588] := 16#5429;
   // UNICODE_TO_GBK[4589] := 16#B7D4;
   // UNICODE_TO_GBK[4590] := 16#542A;
   // UNICODE_TO_GBK[4591] := 16#85C5;
   // UNICODE_TO_GBK[4592] := 16#542B;
   // UNICODE_TO_GBK[4593] := 16#BAAC;
   // UNICODE_TO_GBK[4594] := 16#542C;
   // UNICODE_TO_GBK[4595] := 16#CCFD;
   // UNICODE_TO_GBK[4596] := 16#542D;
   // UNICODE_TO_GBK[4597] := 16#BFD4;
   // UNICODE_TO_GBK[4598] := 16#542E;
   // UNICODE_TO_GBK[4599] := 16#CBB1;
   // UNICODE_TO_GBK[4600] := 16#542F;
   // UNICODE_TO_GBK[4601] := 16#C6F4;
   // UNICODE_TO_GBK[4602] := 16#5430;
   // UNICODE_TO_GBK[4603] := 16#85C6;
   // UNICODE_TO_GBK[4604] := 16#5431;
   // UNICODE_TO_GBK[4605] := 16#D6A8;
   // UNICODE_TO_GBK[4606] := 16#5432;
   // UNICODE_TO_GBK[4607] := 16#DFC5;
   // UNICODE_TO_GBK[4608] := 16#5433;
   // UNICODE_TO_GBK[4609] := 16#85C7;
   // UNICODE_TO_GBK[4610] := 16#5434;
   // UNICODE_TO_GBK[4611] := 16#CEE2;
   // UNICODE_TO_GBK[4612] := 16#5435;
   // UNICODE_TO_GBK[4613] := 16#B3B3;
   // UNICODE_TO_GBK[4614] := 16#5436;
   // UNICODE_TO_GBK[4615] := 16#85C8;
   // UNICODE_TO_GBK[4616] := 16#5437;
   // UNICODE_TO_GBK[4617] := 16#85C9;
   // UNICODE_TO_GBK[4618] := 16#5438;
   // UNICODE_TO_GBK[4619] := 16#CEFC;
   // UNICODE_TO_GBK[4620] := 16#5439;
   // UNICODE_TO_GBK[4621] := 16#B4B5;
   // UNICODE_TO_GBK[4622] := 16#543A;
   // UNICODE_TO_GBK[4623] := 16#85CA;
   // UNICODE_TO_GBK[4624] := 16#543B;
   // UNICODE_TO_GBK[4625] := 16#CEC7;
   // UNICODE_TO_GBK[4626] := 16#543C;
   // UNICODE_TO_GBK[4627] := 16#BAF0;
   // UNICODE_TO_GBK[4628] := 16#543D;
   // UNICODE_TO_GBK[4629] := 16#85CB;
   // UNICODE_TO_GBK[4630] := 16#543E;
   // UNICODE_TO_GBK[4631] := 16#CEE1;
   // UNICODE_TO_GBK[4632] := 16#543F;
   // UNICODE_TO_GBK[4633] := 16#85CC;
   // UNICODE_TO_GBK[4634] := 16#5440;
   // UNICODE_TO_GBK[4635] := 16#D1BD;
   // UNICODE_TO_GBK[4636] := 16#5441;
   // UNICODE_TO_GBK[4637] := 16#85CD;
   // UNICODE_TO_GBK[4638] := 16#5442;
   // UNICODE_TO_GBK[4639] := 16#85CE;
   // UNICODE_TO_GBK[4640] := 16#5443;
   // UNICODE_TO_GBK[4641] := 16#DFC0;
   // UNICODE_TO_GBK[4642] := 16#5444;
   // UNICODE_TO_GBK[4643] := 16#85CF;
   // UNICODE_TO_GBK[4644] := 16#5445;
   // UNICODE_TO_GBK[4645] := 16#85D0;
   // UNICODE_TO_GBK[4646] := 16#5446;
   // UNICODE_TO_GBK[4647] := 16#B4F4;
   // UNICODE_TO_GBK[4648] := 16#5447;
   // UNICODE_TO_GBK[4649] := 16#85D1;
   // UNICODE_TO_GBK[4650] := 16#5448;
   // UNICODE_TO_GBK[4651] := 16#B3CA;
   // UNICODE_TO_GBK[4652] := 16#5449;
   // UNICODE_TO_GBK[4653] := 16#85D2;
   // UNICODE_TO_GBK[4654] := 16#544A;
   // UNICODE_TO_GBK[4655] := 16#B8E6;
   // UNICODE_TO_GBK[4656] := 16#544B;
   // UNICODE_TO_GBK[4657] := 16#DFBB;
   // UNICODE_TO_GBK[4658] := 16#544C;
   // UNICODE_TO_GBK[4659] := 16#85D3;
   // UNICODE_TO_GBK[4660] := 16#544D;
   // UNICODE_TO_GBK[4661] := 16#85D4;
   // UNICODE_TO_GBK[4662] := 16#544E;
   // UNICODE_TO_GBK[4663] := 16#85D5;
   // UNICODE_TO_GBK[4664] := 16#544F;
   // UNICODE_TO_GBK[4665] := 16#85D6;
   // UNICODE_TO_GBK[4666] := 16#5450;
   // UNICODE_TO_GBK[4667] := 16#C4C5;
   // UNICODE_TO_GBK[4668] := 16#5451;
   // UNICODE_TO_GBK[4669] := 16#85D7;
   // UNICODE_TO_GBK[4670] := 16#5452;
   // UNICODE_TO_GBK[4671] := 16#DFBC;
   // UNICODE_TO_GBK[4672] := 16#5453;
   // UNICODE_TO_GBK[4673] := 16#DFBD;
   // UNICODE_TO_GBK[4674] := 16#5454;
   // UNICODE_TO_GBK[4675] := 16#DFBE;
   // UNICODE_TO_GBK[4676] := 16#5455;
   // UNICODE_TO_GBK[4677] := 16#C5BB;
   // UNICODE_TO_GBK[4678] := 16#5456;
   // UNICODE_TO_GBK[4679] := 16#DFBF;
   // UNICODE_TO_GBK[4680] := 16#5457;
   // UNICODE_TO_GBK[4681] := 16#DFC2;
   // UNICODE_TO_GBK[4682] := 16#5458;
   // UNICODE_TO_GBK[4683] := 16#D4B1;
   // UNICODE_TO_GBK[4684] := 16#5459;
   // UNICODE_TO_GBK[4685] := 16#DFC3;
   // UNICODE_TO_GBK[4686] := 16#545A;
   // UNICODE_TO_GBK[4687] := 16#85D8;
   // UNICODE_TO_GBK[4688] := 16#545B;
   // UNICODE_TO_GBK[4689] := 16#C7BA;
   // UNICODE_TO_GBK[4690] := 16#545C;
   // UNICODE_TO_GBK[4691] := 16#CED8;
   // UNICODE_TO_GBK[4692] := 16#545D;
   // UNICODE_TO_GBK[4693] := 16#85D9;
